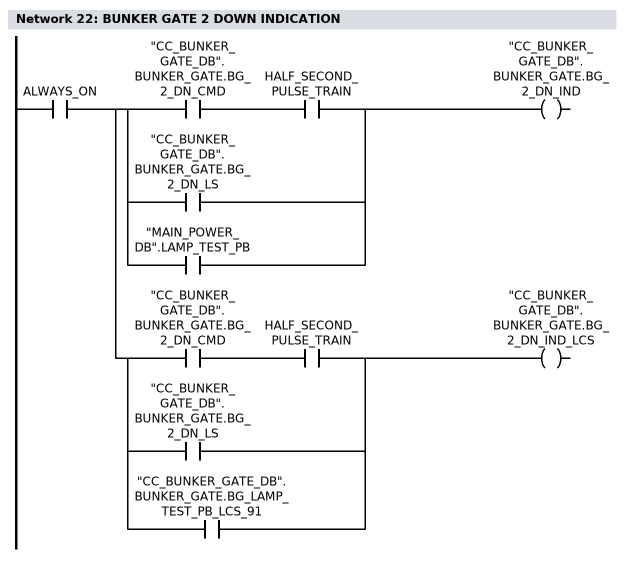
NETWORK
TITLE = BUNKER GATE 2 DOWN INDICATION
      A     "ALWAYS_ON";
      =     L 0.0;
      A     L 0.0;
      A(;
      A     "CC_BUNKER_GATE_DB".BUNKER_GATE.BG_2_DN_CMD;
      A     "HALF_SECOND_PULSE_TRAIN";
      O     "CC_BUNKER_GATE_DB".BUNKER_GATE.BG_2_DN_LS;
      O     "MAIN_POWER_DB".LAMP_TEST_PB;
      );
      =     "CC_BUNKER_GATE_DB".BUNKER_GATE.BG_2_DN_IND;
      A     L 0.0;
      A(;
      A     "CC_BUNKER_GATE_DB".BUNKER_GATE.BG_2_DN_CMD;
      A     "HALF_SECOND_PULSE_TRAIN";
      O     "CC_BUNKER_GATE_DB".BUNKER_GATE.BG_2_DN_LS;
      O     "CC_BUNKER_GATE_DB".BUNKER_GATE.BG_LAMP_TEST_PB_LCS_91;
      );
      =     "CC_BUNKER_GATE_DB".BUNKER_GATE.BG_2_DN_IND_LCS;
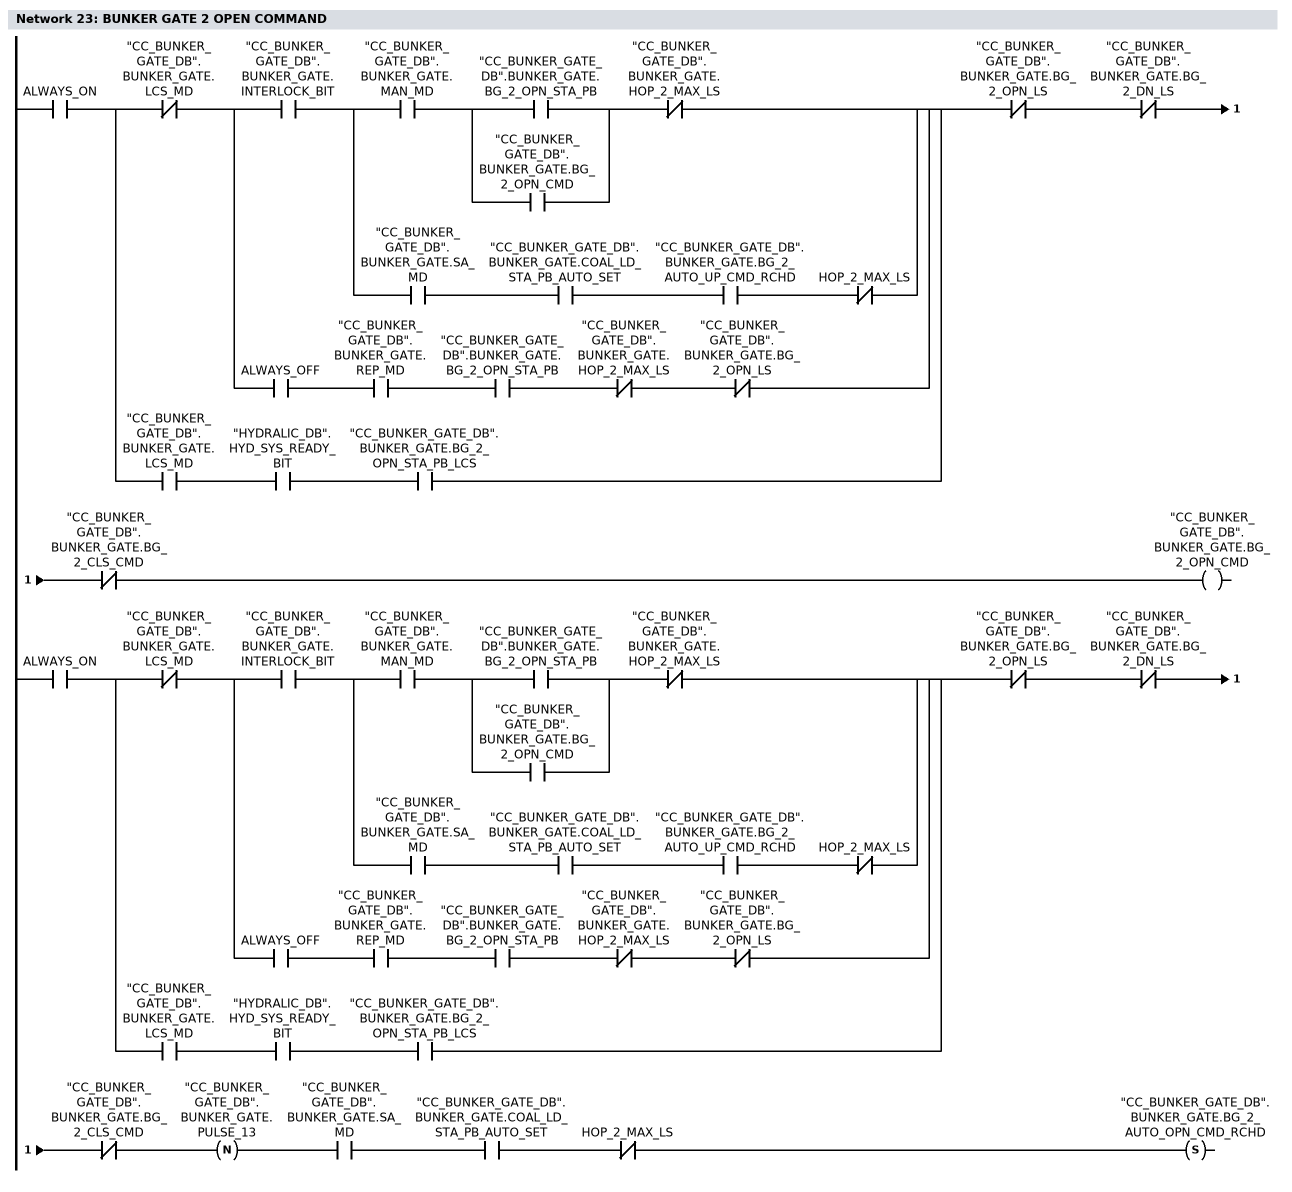
NETWORK
TITLE = BUNKER GATE 2 OPEN COMMAND
      A     "ALWAYS_ON";
      A(;
      AN    "CC_BUNKER_GATE_DB".BUNKER_GATE.LCS_MD;
      A(;
      A     "CC_BUNKER_GATE_DB".BUNKER_GATE.INTERLOCK_BIT;
      A(;
      A     "CC_BUNKER_GATE_DB".BUNKER_GATE.MAN_MD;
      A(;
      O     "CC_BUNKER_GATE_DB".BUNKER_GATE.BG_2_OPN_STA_PB;
      O     "CC_BUNKER_GATE_DB".BUNKER_GATE.BG_2_OPN_CMD;
      );
      AN    "CC_BUNKER_GATE_DB".BUNKER_GATE.HOP_2_MAX_LS;
      O;
      A     "CC_BUNKER_GATE_DB".BUNKER_GATE.SA_MD;
      A     "CC_BUNKER_GATE_DB".BUNKER_GATE.COAL_LD_STA_PB_AUTO_SET;
      A     "CC_BUNKER_GATE_DB".BUNKER_GATE.BG_2_AUTO_UP_CMD_RCHD;
      AN    "HOP_2_MAX_LS";
      );
      O;
      A     "ALWAYS_OFF";
      A     "CC_BUNKER_GATE_DB".BUNKER_GATE.REP_MD;
      A     "CC_BUNKER_GATE_DB".BUNKER_GATE.BG_2_OPN_STA_PB;
      AN    "CC_BUNKER_GATE_DB".BUNKER_GATE.HOP_2_MAX_LS;
      AN    "CC_BUNKER_GATE_DB".BUNKER_GATE.BG_2_OPN_LS;
      );
      O;
      A     "CC_BUNKER_GATE_DB".BUNKER_GATE.LCS_MD;
      A     "HYDRALIC_DB".HYD_SYS_READY_BIT;
      A     "CC_BUNKER_GATE_DB".BUNKER_GATE.BG_2_OPN_STA_PB_LCS;
      );
      AN    "CC_BUNKER_GATE_DB".BUNKER_GATE.BG_2_OPN_LS;
      AN    "CC_BUNKER_GATE_DB".BUNKER_GATE.BG_2_DN_LS;
      AN    "CC_BUNKER_GATE_DB".BUNKER_GATE.BG_2_CLS_CMD;
      =     L 0.0;
      A     L 0.0;
      BLD   102;
      =     "CC_BUNKER_GATE_DB".BUNKER_GATE.BG_2_OPN_CMD;
      A(;
      A     L 0.0;
      FN    "CC_BUNKER_GATE_DB".BUNKER_GATE.PULSE_13;
      );
      A     "CC_BUNKER_GATE_DB".BUNKER_GATE.SA_MD;
      A     "CC_BUNKER_GATE_DB".BUNKER_GATE.COAL_LD_STA_PB_AUTO_SET;
      AN    "HOP_2_MAX_LS";
      S     "CC_BUNKER_GATE_DB".BUNKER_GATE.BG_2_AUTO_OPN_CMD_RCHD;
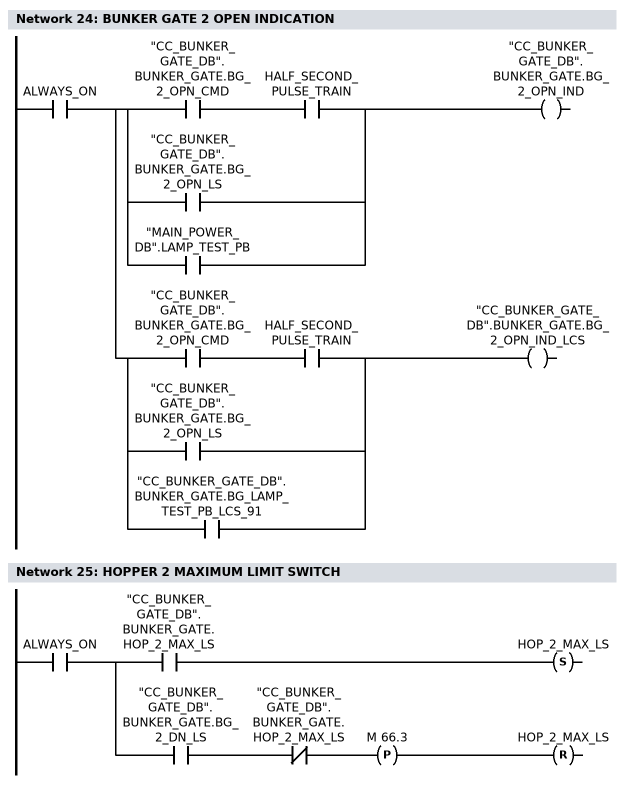
NETWORK
TITLE = BUNKER GATE 2 OPEN INDICATION
      A     "ALWAYS_ON";
      =     L 0.0;
      A     L 0.0;
      A(;
      A     "CC_BUNKER_GATE_DB".BUNKER_GATE.BG_2_OPN_CMD;
      A     "HALF_SECOND_PULSE_TRAIN";
      O     "CC_BUNKER_GATE_DB".BUNKER_GATE.BG_2_OPN_LS;
      O     "MAIN_POWER_DB".LAMP_TEST_PB;
      );
      =     "CC_BUNKER_GATE_DB".BUNKER_GATE.BG_2_OPN_IND;
      A     L 0.0;
      A(;
      A     "CC_BUNKER_GATE_DB".BUNKER_GATE.BG_2_OPN_CMD;
      A     "HALF_SECOND_PULSE_TRAIN";
      O     "CC_BUNKER_GATE_DB".BUNKER_GATE.BG_2_OPN_LS;
      O     "CC_BUNKER_GATE_DB".BUNKER_GATE.BG_LAMP_TEST_PB_LCS_91;
      );
      =     "CC_BUNKER_GATE_DB".BUNKER_GATE.BG_2_OPN_IND_LCS;
NETWORK
TITLE = HOPPER 2 MAXIMUM LIMIT SWITCH
      A     "ALWAYS_ON";
      =     L 0.0;
      A     L 0.0;
      A     "CC_BUNKER_GATE_DB".BUNKER_GATE.HOP_2_MAX_LS;
      S     "HOP_2_MAX_LS";
      A     L 0.0;
      A     "CC_BUNKER_GATE_DB".BUNKER_GATE.BG_2_DN_LS;
      AN    "CC_BUNKER_GATE_DB".BUNKER_GATE.HOP_2_MAX_LS;
      FP    M 66.3;
      R     "HOP_2_MAX_LS";
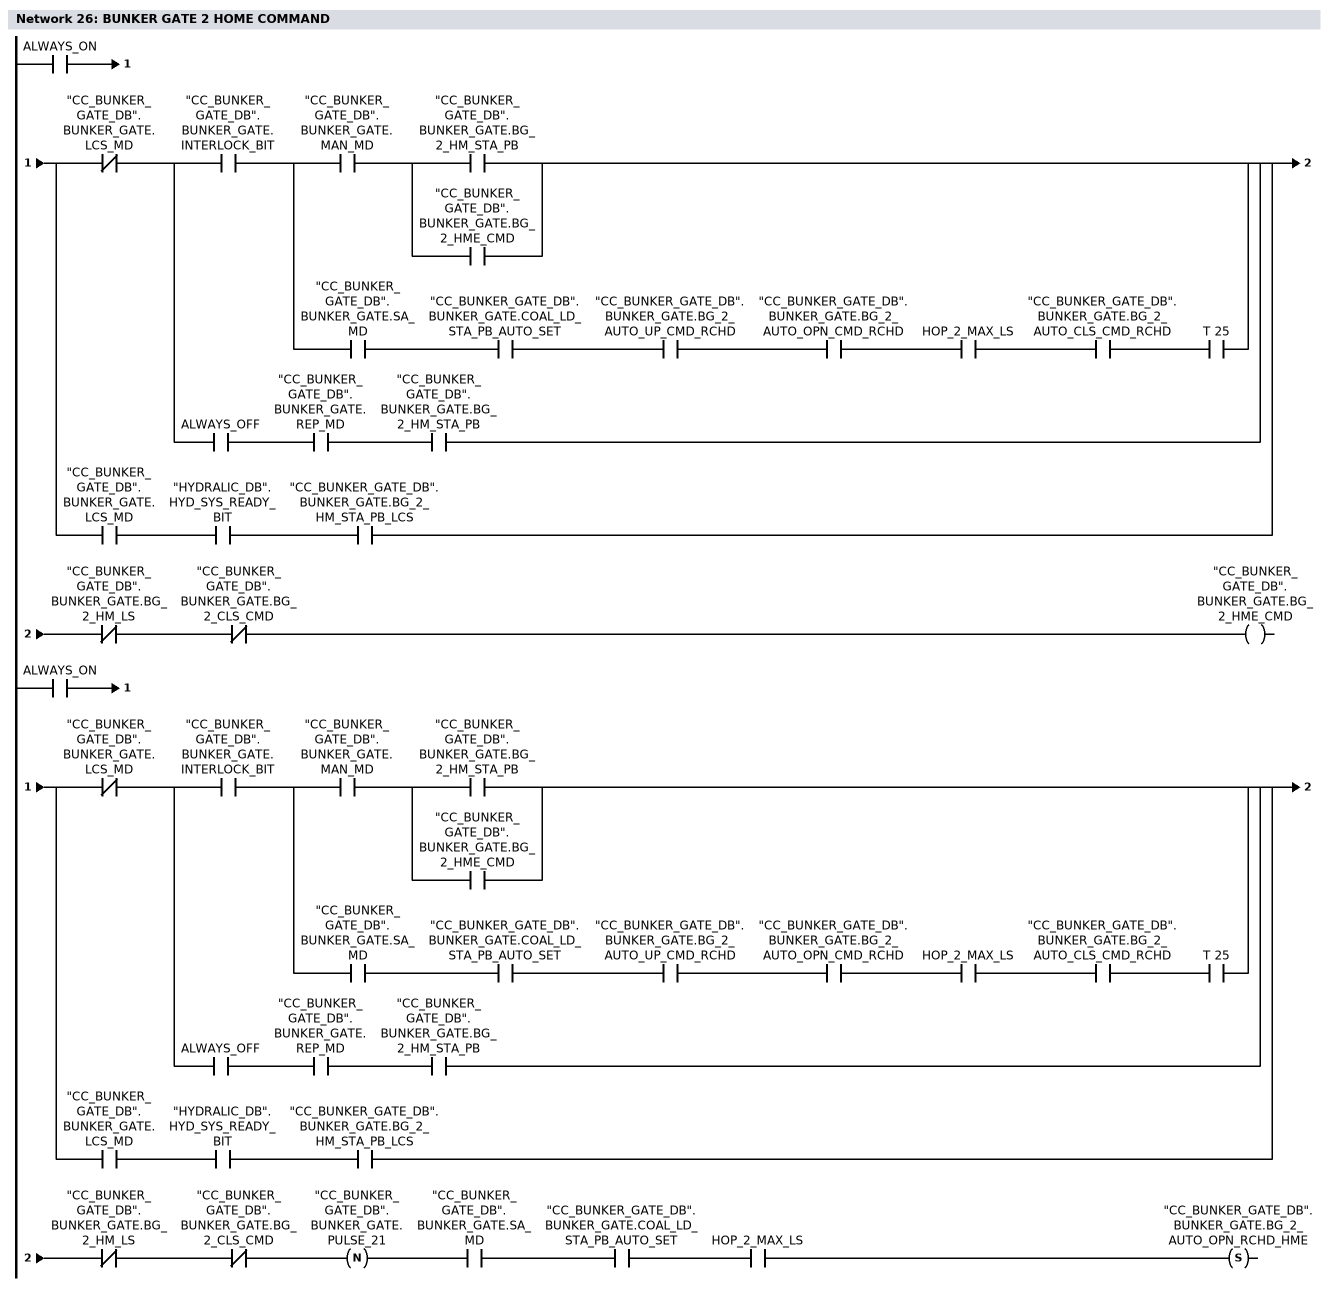
NETWORK
TITLE = BUNKER GATE 2 HOME COMMAND
      A     "ALWAYS_ON";
      A(;
      AN    "CC_BUNKER_GATE_DB".BUNKER_GATE.LCS_MD;
      A(;
      A     "CC_BUNKER_GATE_DB".BUNKER_GATE.INTERLOCK_BIT;
      A(;
      A     "CC_BUNKER_GATE_DB".BUNKER_GATE.MAN_MD;
      A(;
      O     "CC_BUNKER_GATE_DB".BUNKER_GATE.BG_2_HM_STA_PB;
      O     "CC_BUNKER_GATE_DB".BUNKER_GATE.BG_2_HME_CMD;
      );
      O;
      A     "CC_BUNKER_GATE_DB".BUNKER_GATE.SA_MD;
      A     "CC_BUNKER_GATE_DB".BUNKER_GATE.COAL_LD_STA_PB_AUTO_SET;
      A     "CC_BUNKER_GATE_DB".BUNKER_GATE.BG_2_AUTO_UP_CMD_RCHD;
      A     "CC_BUNKER_GATE_DB".BUNKER_GATE.BG_2_AUTO_OPN_CMD_RCHD;
      A     "HOP_2_MAX_LS";
      A     "CC_BUNKER_GATE_DB".BUNKER_GATE.BG_2_AUTO_CLS_CMD_RCHD;
      A     T 25;
      );
      O;
      A     "ALWAYS_OFF";
      A     "CC_BUNKER_GATE_DB".BUNKER_GATE.REP_MD;
      A     "CC_BUNKER_GATE_DB".BUNKER_GATE.BG_2_HM_STA_PB;
      );
      O;
      A     "CC_BUNKER_GATE_DB".BUNKER_GATE.LCS_MD;
      A     "HYDRALIC_DB".HYD_SYS_READY_BIT;
      A     "CC_BUNKER_GATE_DB".BUNKER_GATE.BG_2_HM_STA_PB_LCS;
      );
      AN    "CC_BUNKER_GATE_DB".BUNKER_GATE.BG_2_HM_LS;
      AN    "CC_BUNKER_GATE_DB".BUNKER_GATE.BG_2_CLS_CMD;
      =     L 0.0;
      A     L 0.0;
      BLD   102;
      =     "CC_BUNKER_GATE_DB".BUNKER_GATE.BG_2_HME_CMD;
      A(;
      A     L 0.0;
      FN    "CC_BUNKER_GATE_DB".BUNKER_GATE.PULSE_21;
      );
      A     "CC_BUNKER_GATE_DB".BUNKER_GATE.SA_MD;
      A     "CC_BUNKER_GATE_DB".BUNKER_GATE.COAL_LD_STA_PB_AUTO_SET;
      A     "HOP_2_MAX_LS";
      S     "CC_BUNKER_GATE_DB".BUNKER_GATE.BG_2_AUTO_OPN_RCHD_HME;
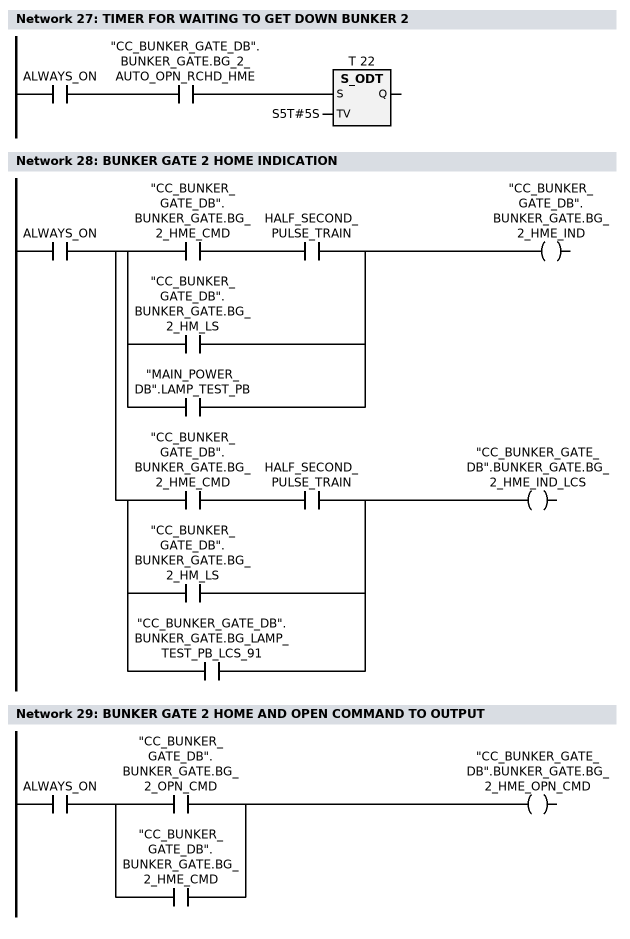
NETWORK
TITLE = TIMER FOR WAITING TO GET DOWN BUNKER 2
      A     "ALWAYS_ON";
      A     "CC_BUNKER_GATE_DB".BUNKER_GATE.BG_2_AUTO_OPN_RCHD_HME;
      L     S5T#5S;
      SD    T 22;
      NOP   0;
      NOP   0;
      NOP   0;
      NOP   0;
NETWORK
TITLE = BUNKER GATE 2 HOME INDICATION
      A     "ALWAYS_ON";
      =     L 0.0;
      A     L 0.0;
      A(;
      A     "CC_BUNKER_GATE_DB".BUNKER_GATE.BG_2_HME_CMD;
      A     "HALF_SECOND_PULSE_TRAIN";
      O     "CC_BUNKER_GATE_DB".BUNKER_GATE.BG_2_HM_LS;
      O     "MAIN_POWER_DB".LAMP_TEST_PB;
      );
      =     "CC_BUNKER_GATE_DB".BUNKER_GATE.BG_2_HME_IND;
      A     L 0.0;
      A(;
      A     "CC_BUNKER_GATE_DB".BUNKER_GATE.BG_2_HME_CMD;
      A     "HALF_SECOND_PULSE_TRAIN";
      O     "CC_BUNKER_GATE_DB".BUNKER_GATE.BG_2_HM_LS;
      O     "CC_BUNKER_GATE_DB".BUNKER_GATE.BG_LAMP_TEST_PB_LCS_91;
      );
      =     "CC_BUNKER_GATE_DB".BUNKER_GATE.BG_2_HME_IND_LCS;
NETWORK
TITLE = BUNKER GATE 2 HOME AND OPEN COMMAND TO OUTPUT
      A     "ALWAYS_ON";
      A(;
      O     "CC_BUNKER_GATE_DB".BUNKER_GATE.BG_2_OPN_CMD;
      O     "CC_BUNKER_GATE_DB".BUNKER_GATE.BG_2_HME_CMD;
      );
      =     "CC_BUNKER_GATE_DB".BUNKER_GATE.BG_2_HME_OPN_CMD;
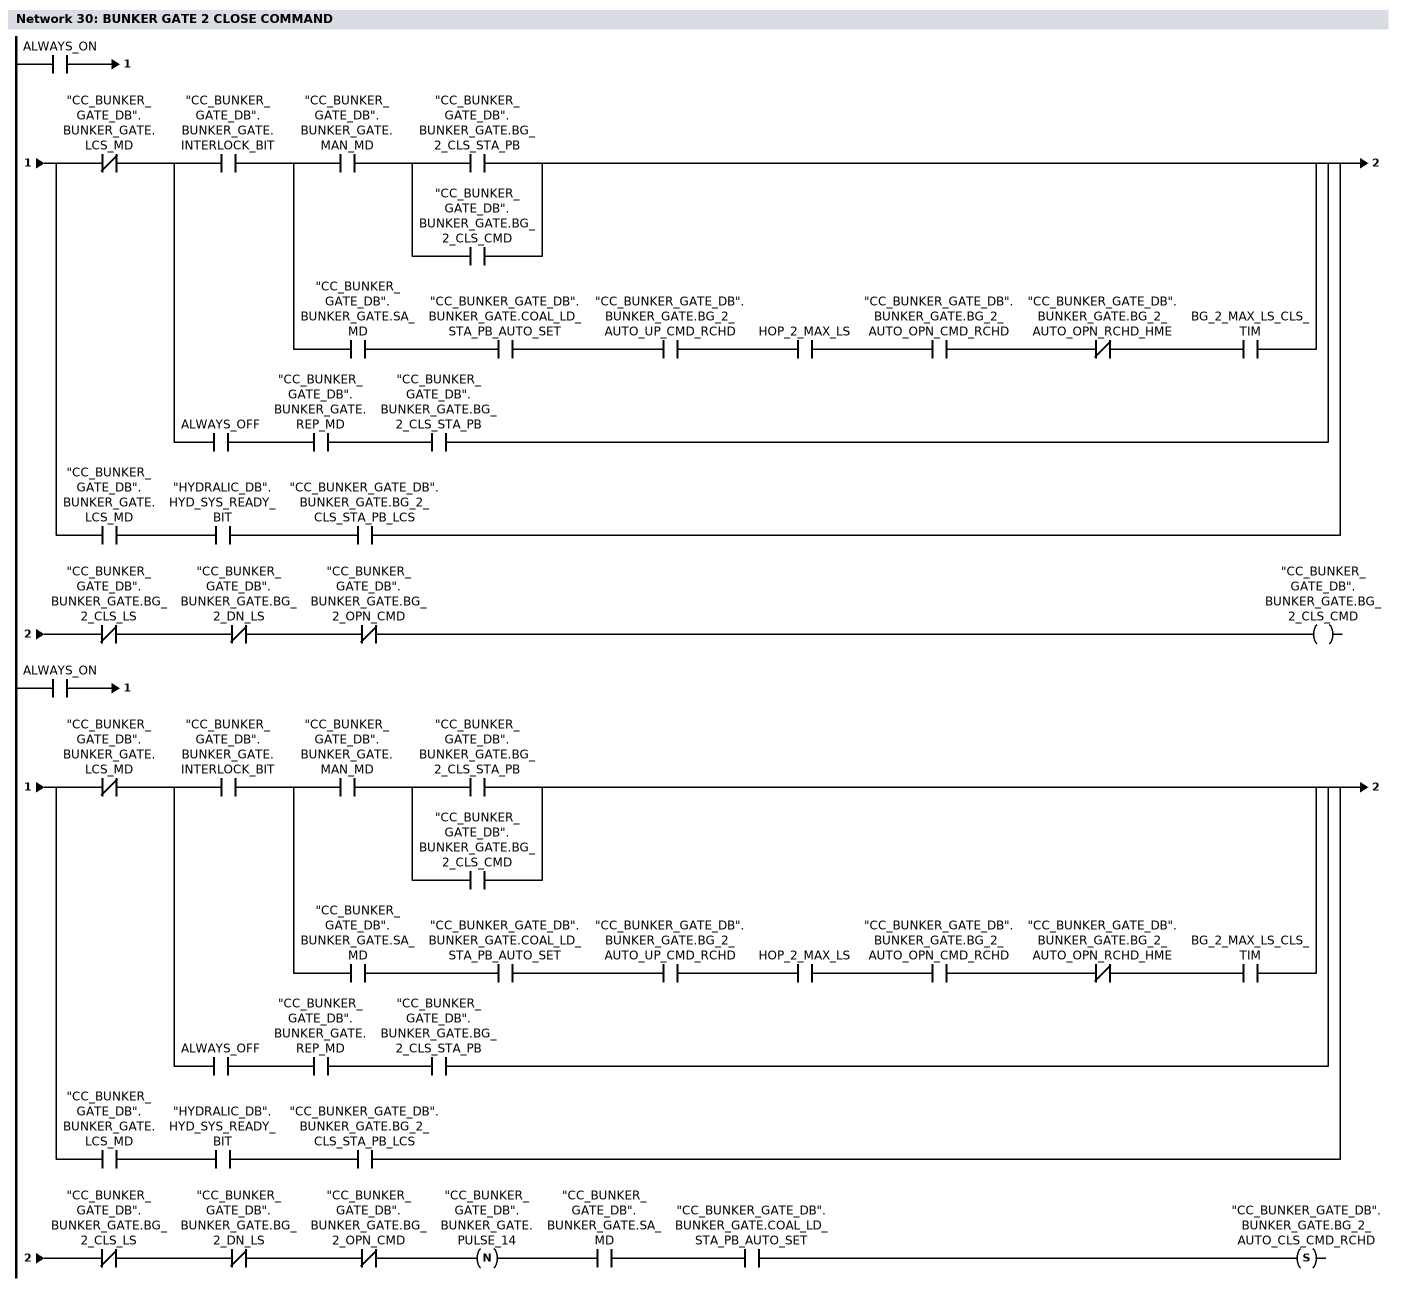
NETWORK
TITLE = BUNKER GATE 2 CLOSE COMMAND
      A     "ALWAYS_ON";
      A(;
      AN    "CC_BUNKER_GATE_DB".BUNKER_GATE.LCS_MD;
      A(;
      A     "CC_BUNKER_GATE_DB".BUNKER_GATE.INTERLOCK_BIT;
      A(;
      A     "CC_BUNKER_GATE_DB".BUNKER_GATE.MAN_MD;
      A(;
      O     "CC_BUNKER_GATE_DB".BUNKER_GATE.BG_2_CLS_STA_PB;
      O     "CC_BUNKER_GATE_DB".BUNKER_GATE.BG_2_CLS_CMD;
      );
      O;
      A     "CC_BUNKER_GATE_DB".BUNKER_GATE.SA_MD;
      A     "CC_BUNKER_GATE_DB".BUNKER_GATE.COAL_LD_STA_PB_AUTO_SET;
      A     "CC_BUNKER_GATE_DB".BUNKER_GATE.BG_2_AUTO_UP_CMD_RCHD;
      A     "HOP_2_MAX_LS";
      A     "CC_BUNKER_GATE_DB".BUNKER_GATE.BG_2_AUTO_OPN_CMD_RCHD;
      AN    "CC_BUNKER_GATE_DB".BUNKER_GATE.BG_2_AUTO_OPN_RCHD_HME;
      A     "BG_2_MAX_LS_CLS_TIM";
      );
      O;
      A     "ALWAYS_OFF";
      A     "CC_BUNKER_GATE_DB".BUNKER_GATE.REP_MD;
      A     "CC_BUNKER_GATE_DB".BUNKER_GATE.BG_2_CLS_STA_PB;
      );
      O;
      A     "CC_BUNKER_GATE_DB".BUNKER_GATE.LCS_MD;
      A     "HYDRALIC_DB".HYD_SYS_READY_BIT;
      A     "CC_BUNKER_GATE_DB".BUNKER_GATE.BG_2_CLS_STA_PB_LCS;
      );
      AN    "CC_BUNKER_GATE_DB".BUNKER_GATE.BG_2_CLS_LS;
      AN    "CC_BUNKER_GATE_DB".BUNKER_GATE.BG_2_DN_LS;
      AN    "CC_BUNKER_GATE_DB".BUNKER_GATE.BG_2_OPN_CMD;
      =     L 0.0;
      A     L 0.0;
      BLD   102;
      =     "CC_BUNKER_GATE_DB".BUNKER_GATE.BG_2_CLS_CMD;
      A(;
      A     L 0.0;
      FN    "CC_BUNKER_GATE_DB".BUNKER_GATE.PULSE_14;
      );
      A     "CC_BUNKER_GATE_DB".BUNKER_GATE.SA_MD;
      A     "CC_BUNKER_GATE_DB".BUNKER_GATE.COAL_LD_STA_PB_AUTO_SET;
      S     "CC_BUNKER_GATE_DB".BUNKER_GATE.BG_2_AUTO_CLS_CMD_RCHD;
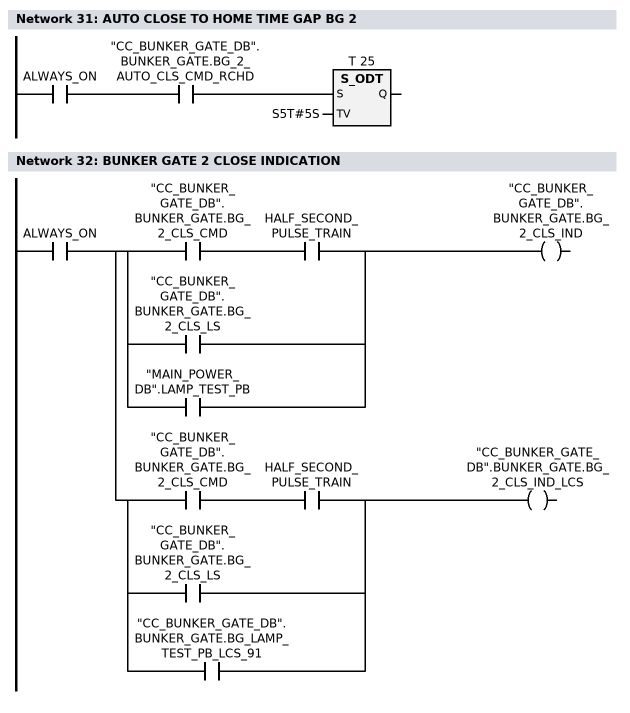
NETWORK
TITLE = AUTO CLOSE TO HOME TIME GAP BG 2
      A     "ALWAYS_ON";
      A     "CC_BUNKER_GATE_DB".BUNKER_GATE.BG_2_AUTO_CLS_CMD_RCHD;
      L     S5T#5S;
      SD    T 25;
      NOP   0;
      NOP   0;
      NOP   0;
      NOP   0;
NETWORK
TITLE = BUNKER GATE 2 CLOSE INDICATION
      A     "ALWAYS_ON";
      =     L 0.0;
      A     L 0.0;
      A(;
      A     "CC_BUNKER_GATE_DB".BUNKER_GATE.BG_2_CLS_CMD;
      A     "HALF_SECOND_PULSE_TRAIN";
      O     "CC_BUNKER_GATE_DB".BUNKER_GATE.BG_2_CLS_LS;
      O     "MAIN_POWER_DB".LAMP_TEST_PB;
      );
      =     "CC_BUNKER_GATE_DB".BUNKER_GATE.BG_2_CLS_IND;
      A     L 0.0;
      A(;
      A     "CC_BUNKER_GATE_DB".BUNKER_GATE.BG_2_CLS_CMD;
      A     "HALF_SECOND_PULSE_TRAIN";
      O     "CC_BUNKER_GATE_DB".BUNKER_GATE.BG_2_CLS_LS;
      O     "CC_BUNKER_GATE_DB".BUNKER_GATE.BG_LAMP_TEST_PB_LCS_91;
      );
      =     "CC_BUNKER_GATE_DB".BUNKER_GATE.BG_2_CLS_IND_LCS;
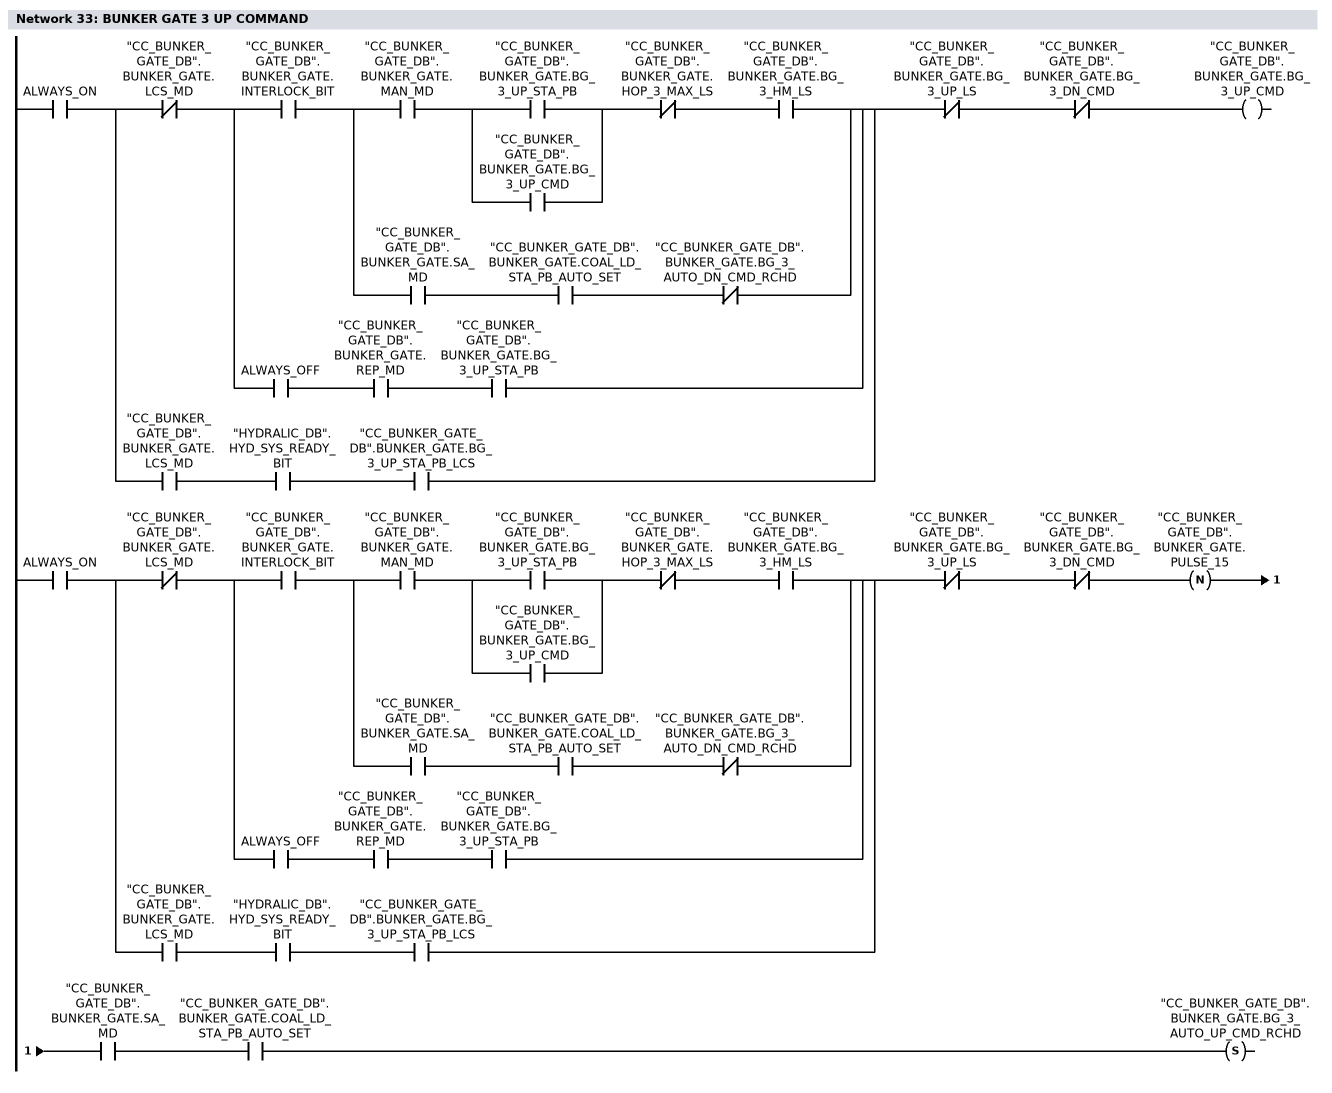
NETWORK
TITLE = BUNKER GATE 3 UP COMMAND
      A     "ALWAYS_ON";
      A(;
      AN    "CC_BUNKER_GATE_DB".BUNKER_GATE.LCS_MD;
      A(;
      A     "CC_BUNKER_GATE_DB".BUNKER_GATE.INTERLOCK_BIT;
      A(;
      A     "CC_BUNKER_GATE_DB".BUNKER_GATE.MAN_MD;
      A(;
      O     "CC_BUNKER_GATE_DB".BUNKER_GATE.BG_3_UP_STA_PB;
      O     "CC_BUNKER_GATE_DB".BUNKER_GATE.BG_3_UP_CMD;
      );
      AN    "CC_BUNKER_GATE_DB".BUNKER_GATE.HOP_3_MAX_LS;
      A     "CC_BUNKER_GATE_DB".BUNKER_GATE.BG_3_HM_LS;
      O;
      A     "CC_BUNKER_GATE_DB".BUNKER_GATE.SA_MD;
      A     "CC_BUNKER_GATE_DB".BUNKER_GATE.COAL_LD_STA_PB_AUTO_SET;
      AN    "CC_BUNKER_GATE_DB".BUNKER_GATE.BG_3_AUTO_DN_CMD_RCHD;
      );
      O;
      A     "ALWAYS_OFF";
      A     "CC_BUNKER_GATE_DB".BUNKER_GATE.REP_MD;
      A     "CC_BUNKER_GATE_DB".BUNKER_GATE.BG_3_UP_STA_PB;
      );
      O;
      A     "CC_BUNKER_GATE_DB".BUNKER_GATE.LCS_MD;
      A     "HYDRALIC_DB".HYD_SYS_READY_BIT;
      A     "CC_BUNKER_GATE_DB".BUNKER_GATE.BG_3_UP_STA_PB_LCS;
      );
      AN    "CC_BUNKER_GATE_DB".BUNKER_GATE.BG_3_UP_LS;
      AN    "CC_BUNKER_GATE_DB".BUNKER_GATE.BG_3_DN_CMD;
      =     L 0.0;
      A     L 0.0;
      BLD   102;
      =     "CC_BUNKER_GATE_DB".BUNKER_GATE.BG_3_UP_CMD;
      A(;
      A     L 0.0;
      FN    "CC_BUNKER_GATE_DB".BUNKER_GATE.PULSE_15;
      );
      A     "CC_BUNKER_GATE_DB".BUNKER_GATE.SA_MD;
      A     "CC_BUNKER_GATE_DB".BUNKER_GATE.COAL_LD_STA_PB_AUTO_SET;
      S     "CC_BUNKER_GATE_DB".BUNKER_GATE.BG_3_AUTO_UP_CMD_RCHD;
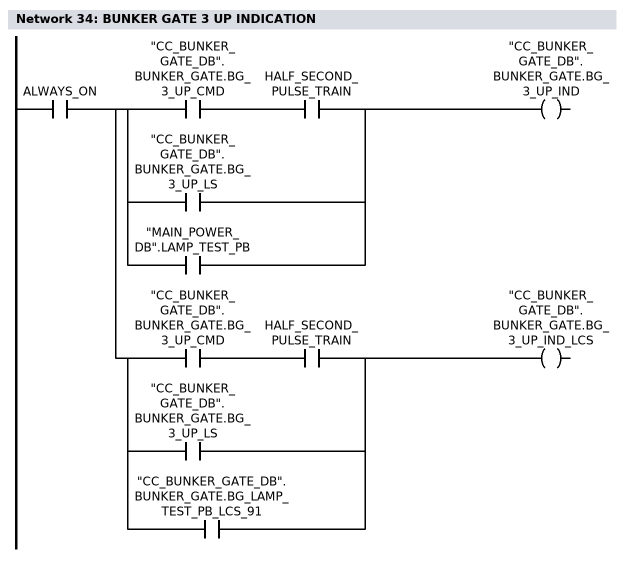
NETWORK
TITLE = BUNKER GATE 3 UP INDICATION
      A     "ALWAYS_ON";
      =     L 0.0;
      A     L 0.0;
      A(;
      A     "CC_BUNKER_GATE_DB".BUNKER_GATE.BG_3_UP_CMD;
      A     "HALF_SECOND_PULSE_TRAIN";
      O     "CC_BUNKER_GATE_DB".BUNKER_GATE.BG_3_UP_LS;
      O     "MAIN_POWER_DB".LAMP_TEST_PB;
      );
      =     "CC_BUNKER_GATE_DB".BUNKER_GATE.BG_3_UP_IND;
      A     L 0.0;
      A(;
      A     "CC_BUNKER_GATE_DB".BUNKER_GATE.BG_3_UP_CMD;
      A     "HALF_SECOND_PULSE_TRAIN";
      O     "CC_BUNKER_GATE_DB".BUNKER_GATE.BG_3_UP_LS;
      O     "CC_BUNKER_GATE_DB".BUNKER_GATE.BG_LAMP_TEST_PB_LCS_91;
      );
      =     "CC_BUNKER_GATE_DB".BUNKER_GATE.BG_3_UP_IND_LCS;
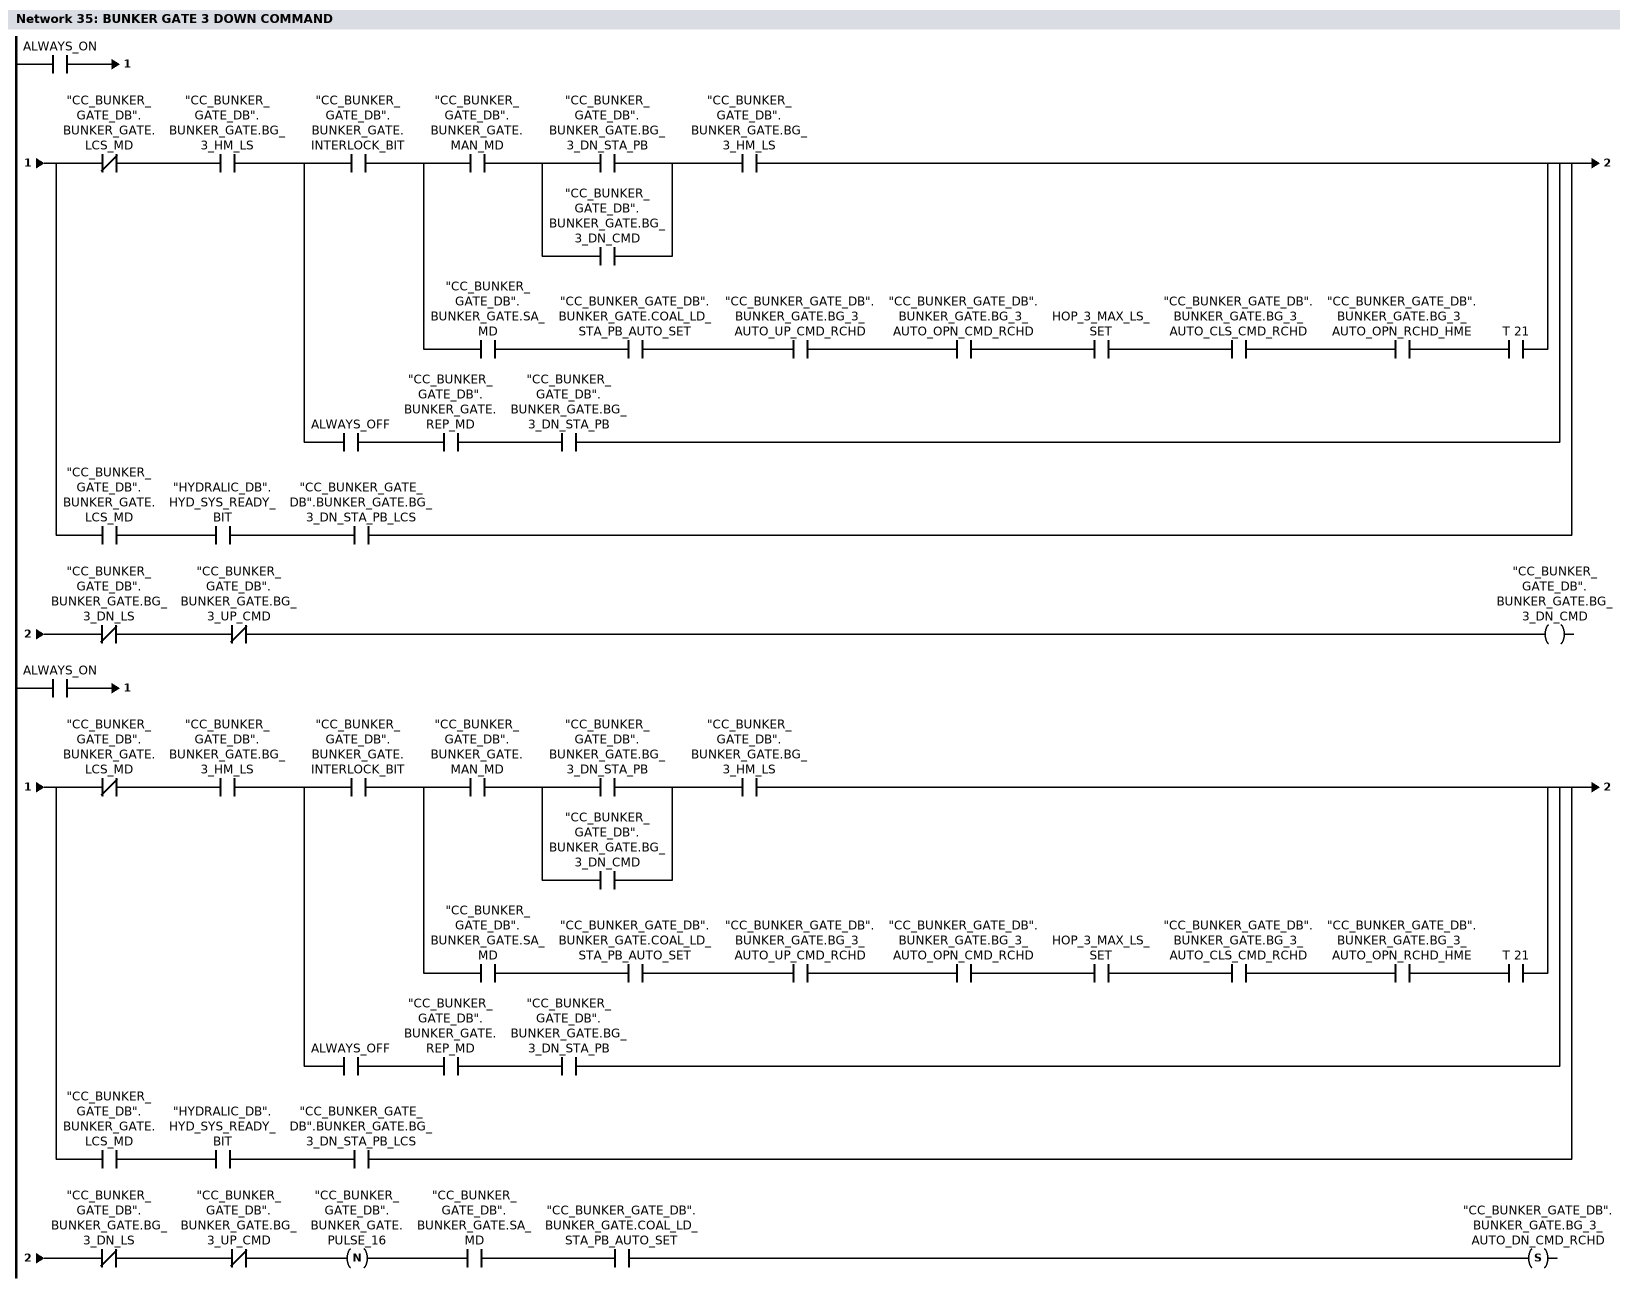
NETWORK
TITLE = BUNKER GATE 3 DOWN COMMAND
      A     "ALWAYS_ON";
      A(;
      AN    "CC_BUNKER_GATE_DB".BUNKER_GATE.LCS_MD;
      A     "CC_BUNKER_GATE_DB".BUNKER_GATE.BG_3_HM_LS;
      A(;
      A     "CC_BUNKER_GATE_DB".BUNKER_GATE.INTERLOCK_BIT;
      A(;
      A     "CC_BUNKER_GATE_DB".BUNKER_GATE.MAN_MD;
      A(;
      O     "CC_BUNKER_GATE_DB".BUNKER_GATE.BG_3_DN_STA_PB;
      O     "CC_BUNKER_GATE_DB".BUNKER_GATE.BG_3_DN_CMD;
      );
      A     "CC_BUNKER_GATE_DB".BUNKER_GATE.BG_3_HM_LS;
      O;
      A     "CC_BUNKER_GATE_DB".BUNKER_GATE.SA_MD;
      A     "CC_BUNKER_GATE_DB".BUNKER_GATE.COAL_LD_STA_PB_AUTO_SET;
      A     "CC_BUNKER_GATE_DB".BUNKER_GATE.BG_3_AUTO_UP_CMD_RCHD;
      A     "CC_BUNKER_GATE_DB".BUNKER_GATE.BG_3_AUTO_OPN_CMD_RCHD;
      A     "HOP_3_MAX_LS_SET";
      A     "CC_BUNKER_GATE_DB".BUNKER_GATE.BG_3_AUTO_CLS_CMD_RCHD;
      A     "CC_BUNKER_GATE_DB".BUNKER_GATE.BG_3_AUTO_OPN_RCHD_HME;
      A     T 21;
      );
      O;
      A     "ALWAYS_OFF";
      A     "CC_BUNKER_GATE_DB".BUNKER_GATE.REP_MD;
      A     "CC_BUNKER_GATE_DB".BUNKER_GATE.BG_3_DN_STA_PB;
      );
      O;
      A     "CC_BUNKER_GATE_DB".BUNKER_GATE.LCS_MD;
      A     "HYDRALIC_DB".HYD_SYS_READY_BIT;
      A     "CC_BUNKER_GATE_DB".BUNKER_GATE.BG_3_DN_STA_PB_LCS;
      );
      AN    "CC_BUNKER_GATE_DB".BUNKER_GATE.BG_3_DN_LS;
      AN    "CC_BUNKER_GATE_DB".BUNKER_GATE.BG_3_UP_CMD;
      =     L 0.0;
      A     L 0.0;
      BLD   102;
      =     "CC_BUNKER_GATE_DB".BUNKER_GATE.BG_3_DN_CMD;
      A(;
      A     L 0.0;
      FN    "CC_BUNKER_GATE_DB".BUNKER_GATE.PULSE_16;
      );
      A     "CC_BUNKER_GATE_DB".BUNKER_GATE.SA_MD;
      A     "CC_BUNKER_GATE_DB".BUNKER_GATE.COAL_LD_STA_PB_AUTO_SET;
      S     "CC_BUNKER_GATE_DB".BUNKER_GATE.BG_3_AUTO_DN_CMD_RCHD;
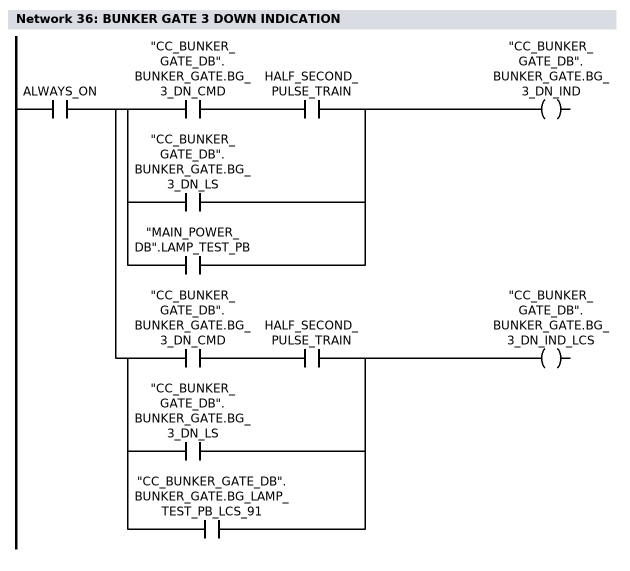
NETWORK
TITLE = BUNKER GATE 3 DOWN INDICATION
      A     "ALWAYS_ON";
      =     L 0.0;
      A     L 0.0;
      A(;
      A     "CC_BUNKER_GATE_DB".BUNKER_GATE.BG_3_DN_CMD;
      A     "HALF_SECOND_PULSE_TRAIN";
      O     "CC_BUNKER_GATE_DB".BUNKER_GATE.BG_3_DN_LS;
      O     "MAIN_POWER_DB".LAMP_TEST_PB;
      );
      =     "CC_BUNKER_GATE_DB".BUNKER_GATE.BG_3_DN_IND;
      A     L 0.0;
      A(;
      A     "CC_BUNKER_GATE_DB".BUNKER_GATE.BG_3_DN_CMD;
      A     "HALF_SECOND_PULSE_TRAIN";
      O     "CC_BUNKER_GATE_DB".BUNKER_GATE.BG_3_DN_LS;
      O     "CC_BUNKER_GATE_DB".BUNKER_GATE.BG_LAMP_TEST_PB_LCS_91;
      );
      =     "CC_BUNKER_GATE_DB".BUNKER_GATE.BG_3_DN_IND_LCS;
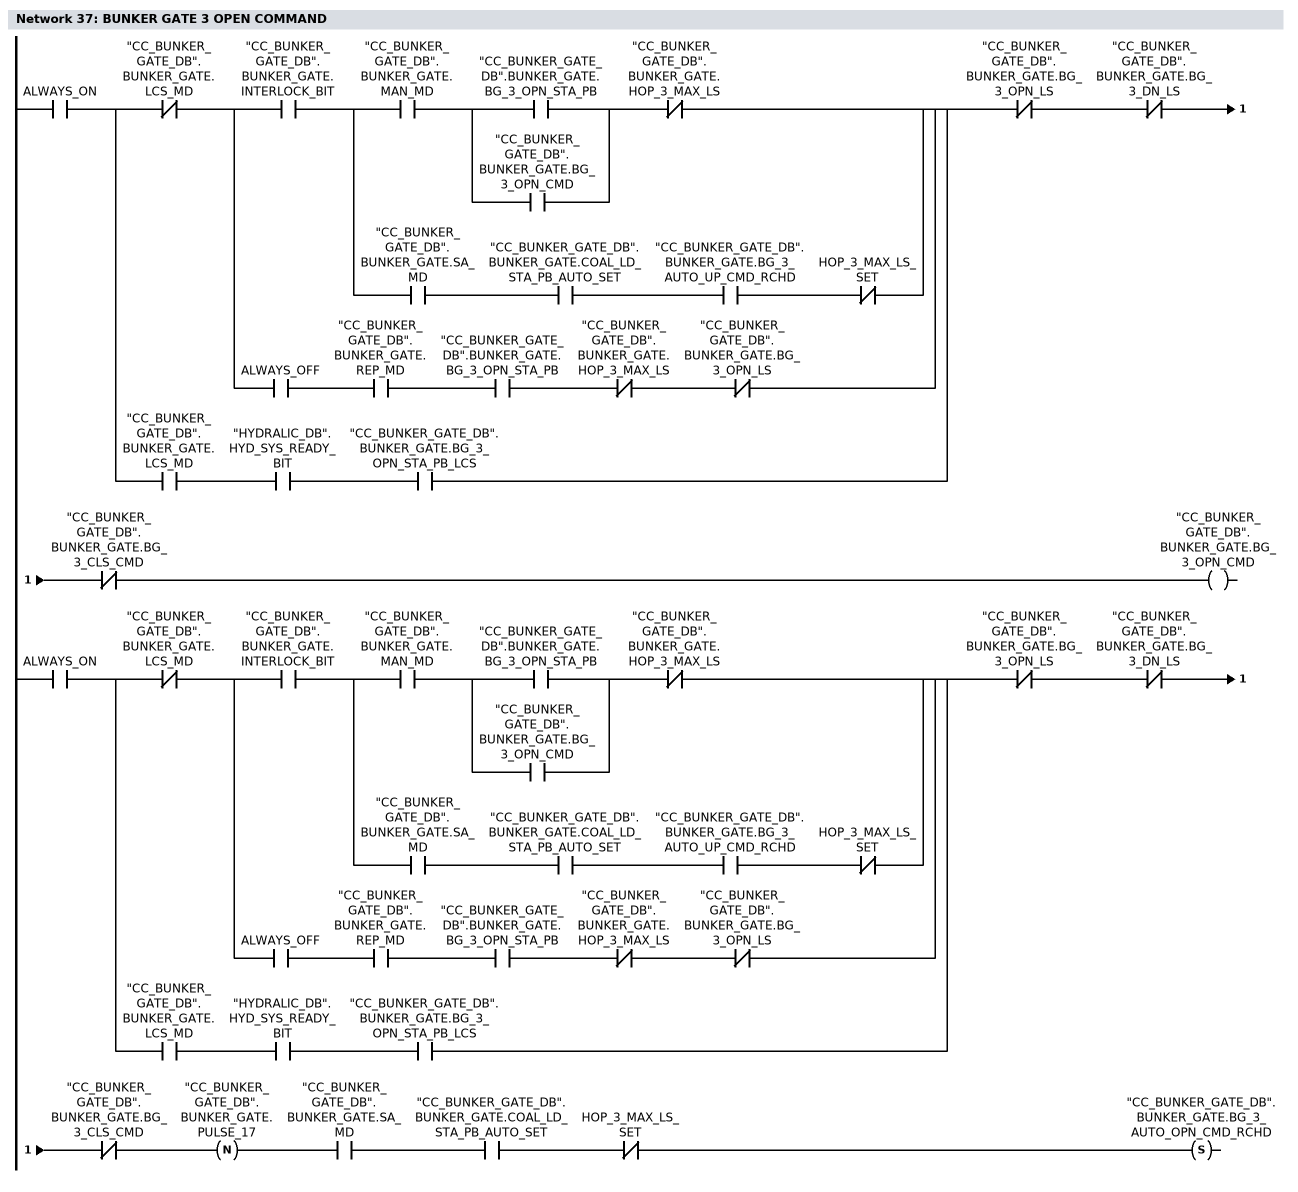
NETWORK
TITLE = BUNKER GATE 3 OPEN COMMAND
      A     "ALWAYS_ON";
      A(;
      AN    "CC_BUNKER_GATE_DB".BUNKER_GATE.LCS_MD;
      A(;
      A     "CC_BUNKER_GATE_DB".BUNKER_GATE.INTERLOCK_BIT;
      A(;
      A     "CC_BUNKER_GATE_DB".BUNKER_GATE.MAN_MD;
      A(;
      O     "CC_BUNKER_GATE_DB".BUNKER_GATE.BG_3_OPN_STA_PB;
      O     "CC_BUNKER_GATE_DB".BUNKER_GATE.BG_3_OPN_CMD;
      );
      AN    "CC_BUNKER_GATE_DB".BUNKER_GATE.HOP_3_MAX_LS;
      O;
      A     "CC_BUNKER_GATE_DB".BUNKER_GATE.SA_MD;
      A     "CC_BUNKER_GATE_DB".BUNKER_GATE.COAL_LD_STA_PB_AUTO_SET;
      A     "CC_BUNKER_GATE_DB".BUNKER_GATE.BG_3_AUTO_UP_CMD_RCHD;
      AN    "HOP_3_MAX_LS_SET";
      );
      O;
      A     "ALWAYS_OFF";
      A     "CC_BUNKER_GATE_DB".BUNKER_GATE.REP_MD;
      A     "CC_BUNKER_GATE_DB".BUNKER_GATE.BG_3_OPN_STA_PB;
      AN    "CC_BUNKER_GATE_DB".BUNKER_GATE.HOP_3_MAX_LS;
      AN    "CC_BUNKER_GATE_DB".BUNKER_GATE.BG_3_OPN_LS;
      );
      O;
      A     "CC_BUNKER_GATE_DB".BUNKER_GATE.LCS_MD;
      A     "HYDRALIC_DB".HYD_SYS_READY_BIT;
      A     "CC_BUNKER_GATE_DB".BUNKER_GATE.BG_3_OPN_STA_PB_LCS;
      );
      AN    "CC_BUNKER_GATE_DB".BUNKER_GATE.BG_3_OPN_LS;
      AN    "CC_BUNKER_GATE_DB".BUNKER_GATE.BG_3_DN_LS;
      AN    "CC_BUNKER_GATE_DB".BUNKER_GATE.BG_3_CLS_CMD;
      =     L 0.0;
      A     L 0.0;
      BLD   102;
      =     "CC_BUNKER_GATE_DB".BUNKER_GATE.BG_3_OPN_CMD;
      A(;
      A     L 0.0;
      FN    "CC_BUNKER_GATE_DB".BUNKER_GATE.PULSE_17;
      );
      A     "CC_BUNKER_GATE_DB".BUNKER_GATE.SA_MD;
      A     "CC_BUNKER_GATE_DB".BUNKER_GATE.COAL_LD_STA_PB_AUTO_SET;
      AN    "HOP_3_MAX_LS_SET";
      S     "CC_BUNKER_GATE_DB".BUNKER_GATE.BG_3_AUTO_OPN_CMD_RCHD;
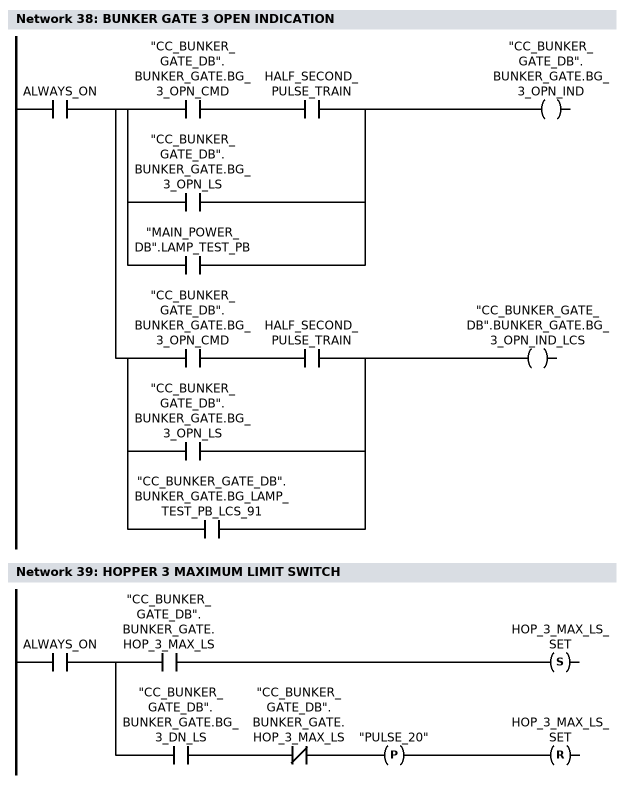
NETWORK
TITLE = BUNKER GATE 3 OPEN INDICATION
      A     "ALWAYS_ON";
      =     L 0.0;
      A     L 0.0;
      A(;
      A     "CC_BUNKER_GATE_DB".BUNKER_GATE.BG_3_OPN_CMD;
      A     "HALF_SECOND_PULSE_TRAIN";
      O     "CC_BUNKER_GATE_DB".BUNKER_GATE.BG_3_OPN_LS;
      O     "MAIN_POWER_DB".LAMP_TEST_PB;
      );
      =     "CC_BUNKER_GATE_DB".BUNKER_GATE.BG_3_OPN_IND;
      A     L 0.0;
      A(;
      A     "CC_BUNKER_GATE_DB".BUNKER_GATE.BG_3_OPN_CMD;
      A     "HALF_SECOND_PULSE_TRAIN";
      O     "CC_BUNKER_GATE_DB".BUNKER_GATE.BG_3_OPN_LS;
      O     "CC_BUNKER_GATE_DB".BUNKER_GATE.BG_LAMP_TEST_PB_LCS_91;
      );
      =     "CC_BUNKER_GATE_DB".BUNKER_GATE.BG_3_OPN_IND_LCS;
NETWORK
TITLE = HOPPER 3 MAXIMUM LIMIT SWITCH
      A     "ALWAYS_ON";
      =     L 0.0;
      A     L 0.0;
      A     "CC_BUNKER_GATE_DB".BUNKER_GATE.HOP_3_MAX_LS;
      S     "HOP_3_MAX_LS_SET";
      A     L 0.0;
      A     "CC_BUNKER_GATE_DB".BUNKER_GATE.BG_3_DN_LS;
      AN    "CC_BUNKER_GATE_DB".BUNKER_GATE.HOP_3_MAX_LS;
      FP    "PULSE_20";
      R     "HOP_3_MAX_LS_SET";
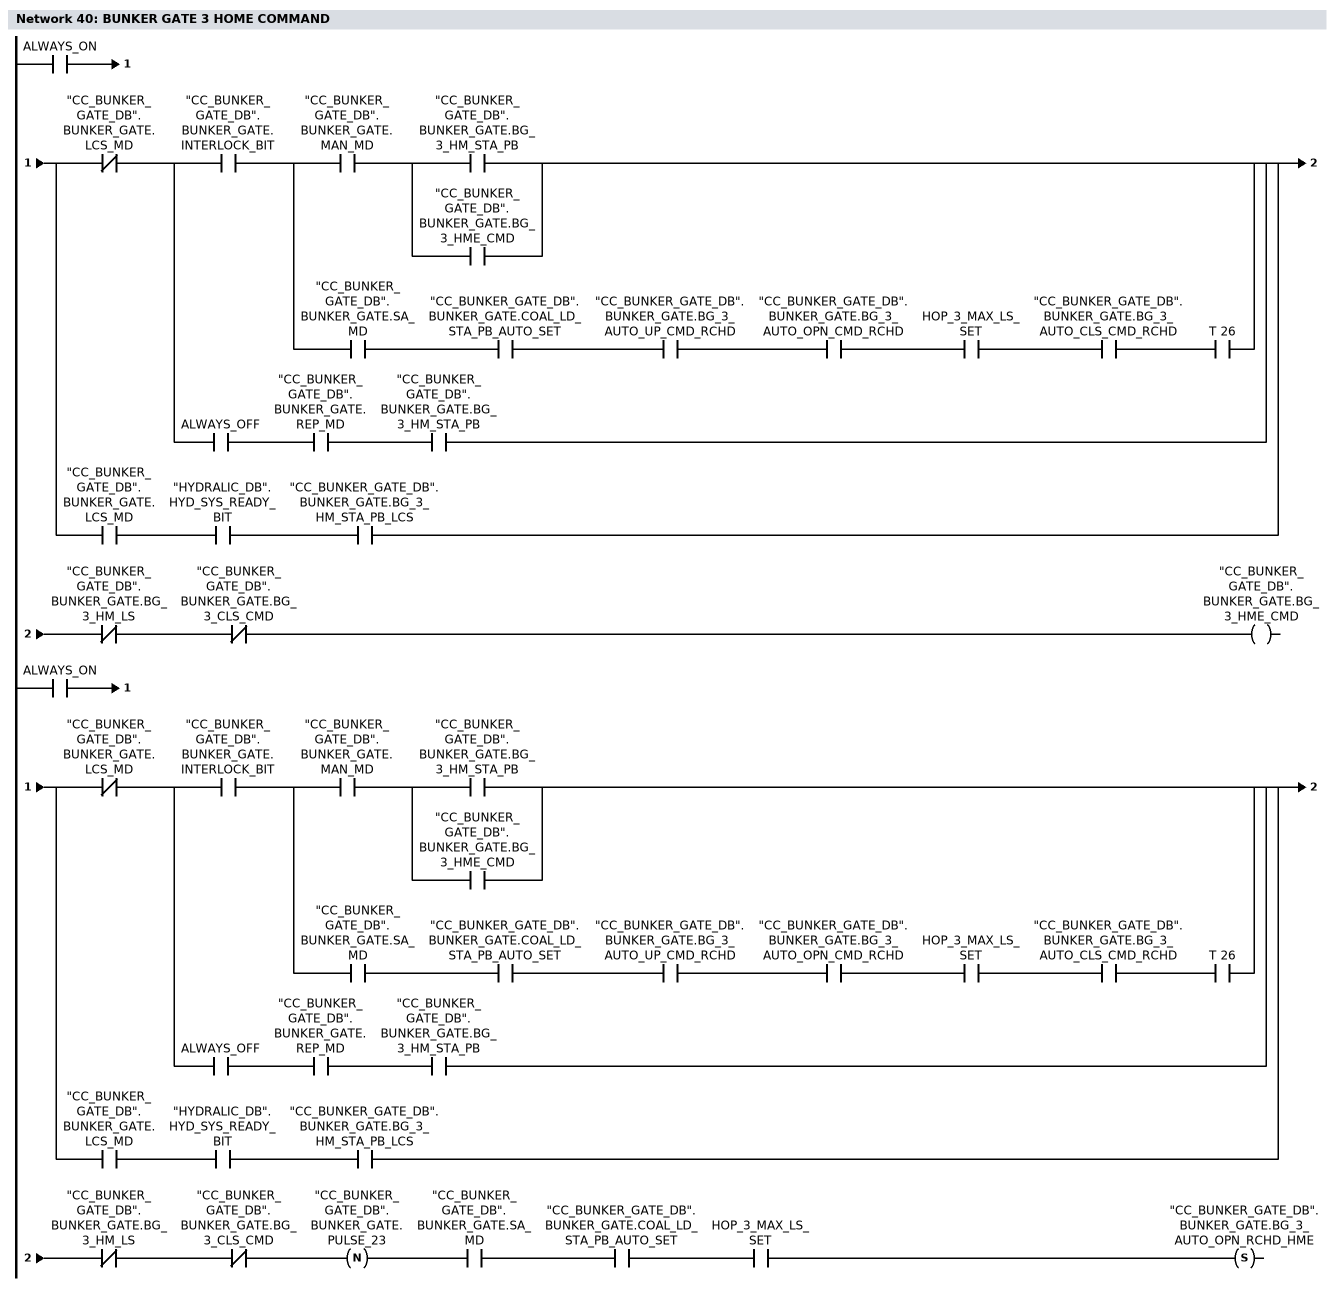
NETWORK
TITLE = BUNKER GATE 3 HOME COMMAND
      A     "ALWAYS_ON";
      A(;
      AN    "CC_BUNKER_GATE_DB".BUNKER_GATE.LCS_MD;
      A(;
      A     "CC_BUNKER_GATE_DB".BUNKER_GATE.INTERLOCK_BIT;
      A(;
      A     "CC_BUNKER_GATE_DB".BUNKER_GATE.MAN_MD;
      A(;
      O     "CC_BUNKER_GATE_DB".BUNKER_GATE.BG_3_HM_STA_PB;
      O     "CC_BUNKER_GATE_DB".BUNKER_GATE.BG_3_HME_CMD;
      );
      O;
      A     "CC_BUNKER_GATE_DB".BUNKER_GATE.SA_MD;
      A     "CC_BUNKER_GATE_DB".BUNKER_GATE.COAL_LD_STA_PB_AUTO_SET;
      A     "CC_BUNKER_GATE_DB".BUNKER_GATE.BG_3_AUTO_UP_CMD_RCHD;
      A     "CC_BUNKER_GATE_DB".BUNKER_GATE.BG_3_AUTO_OPN_CMD_RCHD;
      A     "HOP_3_MAX_LS_SET";
      A     "CC_BUNKER_GATE_DB".BUNKER_GATE.BG_3_AUTO_CLS_CMD_RCHD;
      A     T 26;
      );
      O;
      A     "ALWAYS_OFF";
      A     "CC_BUNKER_GATE_DB".BUNKER_GATE.REP_MD;
      A     "CC_BUNKER_GATE_DB".BUNKER_GATE.BG_3_HM_STA_PB;
      );
      O;
      A     "CC_BUNKER_GATE_DB".BUNKER_GATE.LCS_MD;
      A     "HYDRALIC_DB".HYD_SYS_READY_BIT;
      A     "CC_BUNKER_GATE_DB".BUNKER_GATE.BG_3_HM_STA_PB_LCS;
      );
      AN    "CC_BUNKER_GATE_DB".BUNKER_GATE.BG_3_HM_LS;
      AN    "CC_BUNKER_GATE_DB".BUNKER_GATE.BG_3_CLS_CMD;
      =     L 0.0;
      A     L 0.0;
      BLD   102;
      =     "CC_BUNKER_GATE_DB".BUNKER_GATE.BG_3_HME_CMD;
      A(;
      A     L 0.0;
      FN    "CC_BUNKER_GATE_DB".BUNKER_GATE.PULSE_23;
      );
      A     "CC_BUNKER_GATE_DB".BUNKER_GATE.SA_MD;
      A     "CC_BUNKER_GATE_DB".BUNKER_GATE.COAL_LD_STA_PB_AUTO_SET;
      A     "HOP_3_MAX_LS_SET";
      S     "CC_BUNKER_GATE_DB".BUNKER_GATE.BG_3_AUTO_OPN_RCHD_HME;
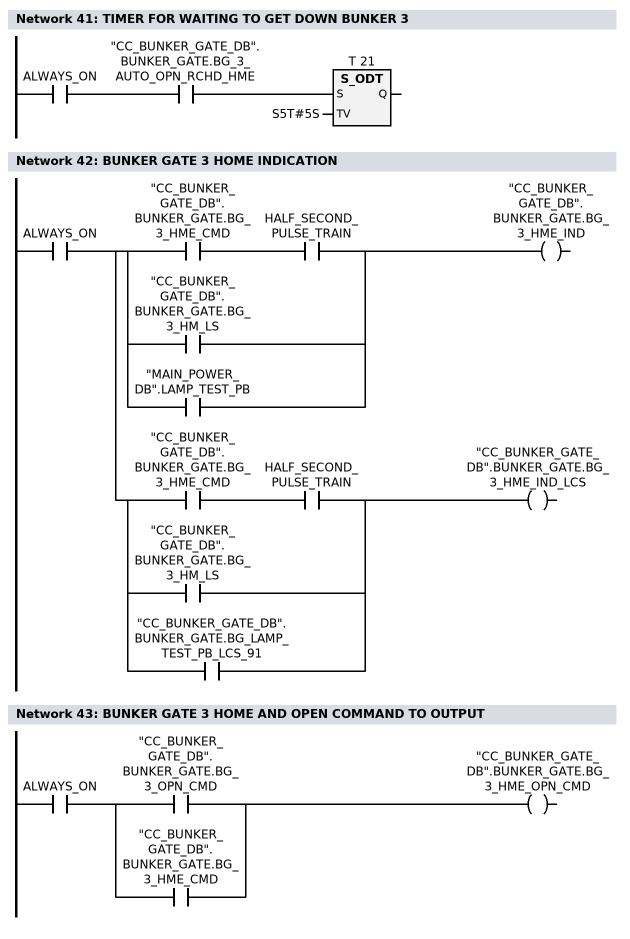
NETWORK
TITLE = TIMER FOR WAITING TO GET DOWN BUNKER 3
      A     "ALWAYS_ON";
      A     "CC_BUNKER_GATE_DB".BUNKER_GATE.BG_3_AUTO_OPN_RCHD_HME;
      L     S5T#5S;
      SD    T 21;
      NOP   0;
      NOP   0;
      NOP   0;
      NOP   0;
NETWORK
TITLE = BUNKER GATE 3 HOME INDICATION
      A     "ALWAYS_ON";
      =     L 0.0;
      A     L 0.0;
      A(;
      A     "CC_BUNKER_GATE_DB".BUNKER_GATE.BG_3_HME_CMD;
      A     "HALF_SECOND_PULSE_TRAIN";
      O     "CC_BUNKER_GATE_DB".BUNKER_GATE.BG_3_HM_LS;
      O     "MAIN_POWER_DB".LAMP_TEST_PB;
      );
      =     "CC_BUNKER_GATE_DB".BUNKER_GATE.BG_3_HME_IND;
      A     L 0.0;
      A(;
      A     "CC_BUNKER_GATE_DB".BUNKER_GATE.BG_3_HME_CMD;
      A     "HALF_SECOND_PULSE_TRAIN";
      O     "CC_BUNKER_GATE_DB".BUNKER_GATE.BG_3_HM_LS;
      O     "CC_BUNKER_GATE_DB".BUNKER_GATE.BG_LAMP_TEST_PB_LCS_91;
      );
      =     "CC_BUNKER_GATE_DB".BUNKER_GATE.BG_3_HME_IND_LCS;
NETWORK
TITLE = BUNKER GATE 3 HOME AND OPEN COMMAND TO OUTPUT
      A     "ALWAYS_ON";
      A(;
      O     "CC_BUNKER_GATE_DB".BUNKER_GATE.BG_3_OPN_CMD;
      O     "CC_BUNKER_GATE_DB".BUNKER_GATE.BG_3_HME_CMD;
      );
      =     "CC_BUNKER_GATE_DB".BUNKER_GATE.BG_3_HME_OPN_CMD;
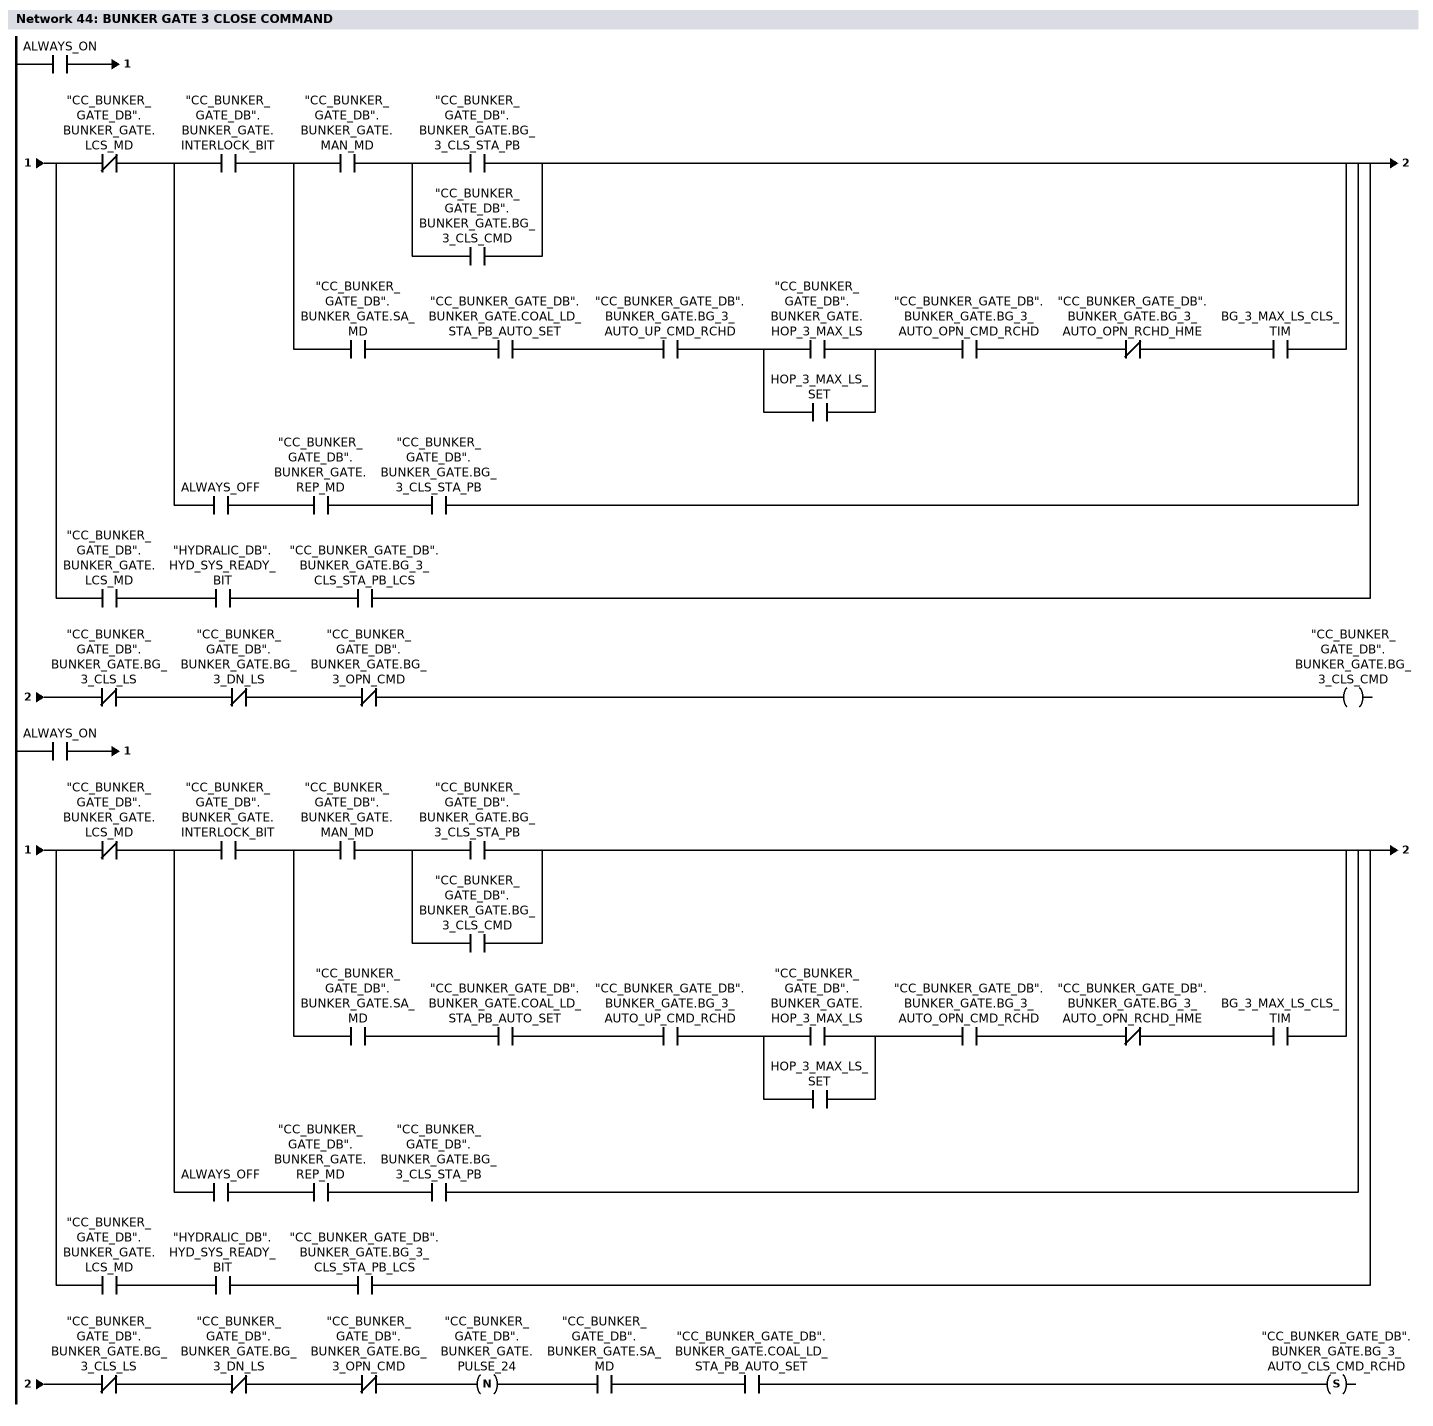
NETWORK
TITLE = BUNKER GATE 3 CLOSE COMMAND
      A     "ALWAYS_ON";
      A(;
      AN    "CC_BUNKER_GATE_DB".BUNKER_GATE.LCS_MD;
      A(;
      A     "CC_BUNKER_GATE_DB".BUNKER_GATE.INTERLOCK_BIT;
      A(;
      A     "CC_BUNKER_GATE_DB".BUNKER_GATE.MAN_MD;
      A(;
      O     "CC_BUNKER_GATE_DB".BUNKER_GATE.BG_3_CLS_STA_PB;
      O     "CC_BUNKER_GATE_DB".BUNKER_GATE.BG_3_CLS_CMD;
      );
      O;
      A     "CC_BUNKER_GATE_DB".BUNKER_GATE.SA_MD;
      A     "CC_BUNKER_GATE_DB".BUNKER_GATE.COAL_LD_STA_PB_AUTO_SET;
      A     "CC_BUNKER_GATE_DB".BUNKER_GATE.BG_3_AUTO_UP_CMD_RCHD;
      A(;
      O     "CC_BUNKER_GATE_DB".BUNKER_GATE.HOP_3_MAX_LS;
      O     "HOP_3_MAX_LS_SET";
      );
      A     "CC_BUNKER_GATE_DB".BUNKER_GATE.BG_3_AUTO_OPN_CMD_RCHD;
      AN    "CC_BUNKER_GATE_DB".BUNKER_GATE.BG_3_AUTO_OPN_RCHD_HME;
      A     "BG_3_MAX_LS_CLS_TIM";
      );
      O;
      A     "ALWAYS_OFF";
      A     "CC_BUNKER_GATE_DB".BUNKER_GATE.REP_MD;
      A     "CC_BUNKER_GATE_DB".BUNKER_GATE.BG_3_CLS_STA_PB;
      );
      O;
      A     "CC_BUNKER_GATE_DB".BUNKER_GATE.LCS_MD;
      A     "HYDRALIC_DB".HYD_SYS_READY_BIT;
      A     "CC_BUNKER_GATE_DB".BUNKER_GATE.BG_3_CLS_STA_PB_LCS;
      );
      AN    "CC_BUNKER_GATE_DB".BUNKER_GATE.BG_3_CLS_LS;
      AN    "CC_BUNKER_GATE_DB".BUNKER_GATE.BG_3_DN_LS;
      AN    "CC_BUNKER_GATE_DB".BUNKER_GATE.BG_3_OPN_CMD;
      =     L 0.0;
      A     L 0.0;
      BLD   102;
      =     "CC_BUNKER_GATE_DB".BUNKER_GATE.BG_3_CLS_CMD;
      A(;
      A     L 0.0;
      FN    "CC_BUNKER_GATE_DB".BUNKER_GATE.PULSE_24;
      );
      A     "CC_BUNKER_GATE_DB".BUNKER_GATE.SA_MD;
      A     "CC_BUNKER_GATE_DB".BUNKER_GATE.COAL_LD_STA_PB_AUTO_SET;
      S     "CC_BUNKER_GATE_DB".BUNKER_GATE.BG_3_AUTO_CLS_CMD_RCHD;
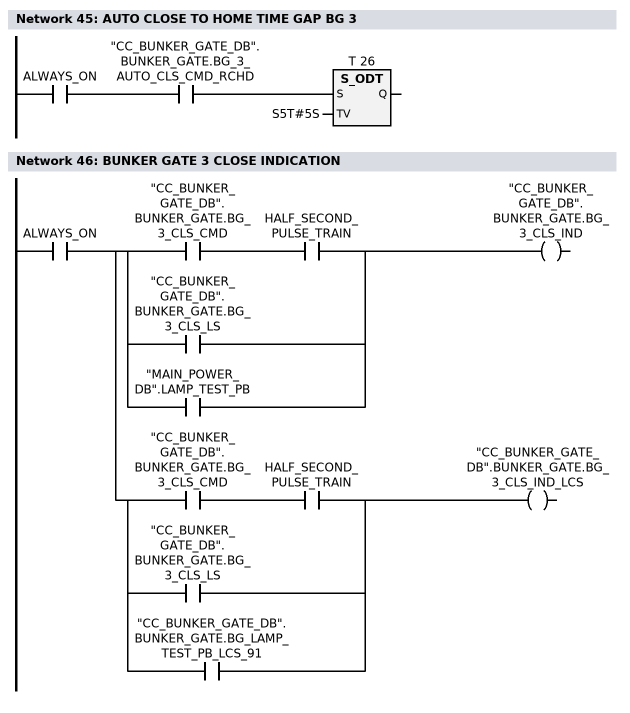
NETWORK
TITLE = AUTO CLOSE TO HOME TIME GAP BG 3
      A     "ALWAYS_ON";
      A     "CC_BUNKER_GATE_DB".BUNKER_GATE.BG_3_AUTO_CLS_CMD_RCHD;
      L     S5T#5S;
      SD    T 26;
      NOP   0;
      NOP   0;
      NOP   0;
      NOP   0;
NETWORK
TITLE = BUNKER GATE 3 CLOSE INDICATION
      A     "ALWAYS_ON";
      =     L 0.0;
      A     L 0.0;
      A(;
      A     "CC_BUNKER_GATE_DB".BUNKER_GATE.BG_3_CLS_CMD;
      A     "HALF_SECOND_PULSE_TRAIN";
      O     "CC_BUNKER_GATE_DB".BUNKER_GATE.BG_3_CLS_LS;
      O     "MAIN_POWER_DB".LAMP_TEST_PB;
      );
      =     "CC_BUNKER_GATE_DB".BUNKER_GATE.BG_3_CLS_IND;
      A     L 0.0;
      A(;
      A     "CC_BUNKER_GATE_DB".BUNKER_GATE.BG_3_CLS_CMD;
      A     "HALF_SECOND_PULSE_TRAIN";
      O     "CC_BUNKER_GATE_DB".BUNKER_GATE.BG_3_CLS_LS;
      O     "CC_BUNKER_GATE_DB".BUNKER_GATE.BG_LAMP_TEST_PB_LCS_91;
      );
      =     "CC_BUNKER_GATE_DB".BUNKER_GATE.BG_3_CLS_IND_LCS;
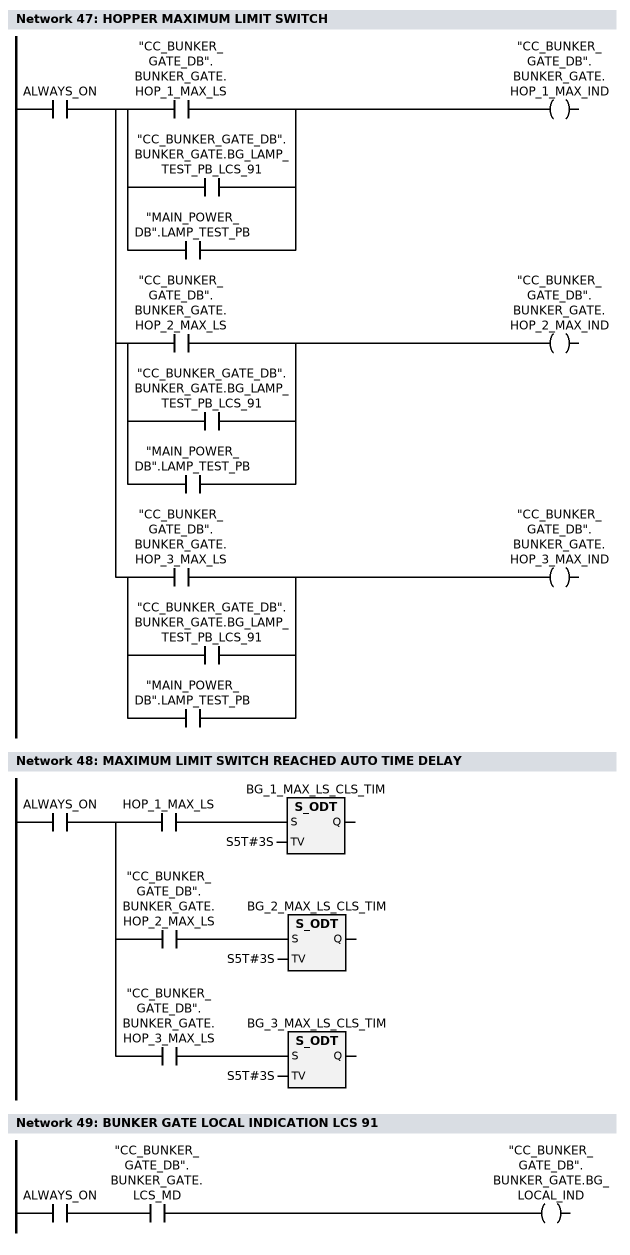
NETWORK
TITLE = HOPPER MAXIMUM LIMIT SWITCH
      A     "ALWAYS_ON";
      =     L 0.0;
      A     L 0.0;
      A(;
      O     "CC_BUNKER_GATE_DB".BUNKER_GATE.HOP_1_MAX_LS;
      O     "CC_BUNKER_GATE_DB".BUNKER_GATE.BG_LAMP_TEST_PB_LCS_91;
      O     "MAIN_POWER_DB".LAMP_TEST_PB;
      );
      =     "CC_BUNKER_GATE_DB".BUNKER_GATE.HOP_1_MAX_IND;
      A     L 0.0;
      A(;
      O     "CC_BUNKER_GATE_DB".BUNKER_GATE.HOP_2_MAX_LS;
      O     "CC_BUNKER_GATE_DB".BUNKER_GATE.BG_LAMP_TEST_PB_LCS_91;
      O     "MAIN_POWER_DB".LAMP_TEST_PB;
      );
      =     "CC_BUNKER_GATE_DB".BUNKER_GATE.HOP_2_MAX_IND;
      A     L 0.0;
      A(;
      O     "CC_BUNKER_GATE_DB".BUNKER_GATE.HOP_3_MAX_LS;
      O     "CC_BUNKER_GATE_DB".BUNKER_GATE.BG_LAMP_TEST_PB_LCS_91;
      O     "MAIN_POWER_DB".LAMP_TEST_PB;
      );
      =     "CC_BUNKER_GATE_DB".BUNKER_GATE.HOP_3_MAX_IND;
NETWORK
TITLE = MAXIMUM LIMIT SWITCH REACHED AUTO TIME DELAY
      A     "ALWAYS_ON";
      =     L 0.0;
      A     L 0.0;
      A     "HOP_1_MAX_LS";
      L     S5T#3S;
      SD    "BG_1_MAX_LS_CLS_TIM";
      NOP   0;
      NOP   0;
      NOP   0;
      NOP   0;
      A     L 0.0;
      A     "CC_BUNKER_GATE_DB".BUNKER_GATE.HOP_2_MAX_LS;
      L     S5T#3S;
      SD    "BG_2_MAX_LS_CLS_TIM";
      NOP   0;
      NOP   0;
      NOP   0;
      NOP   0;
      A     L 0.0;
      A     "CC_BUNKER_GATE_DB".BUNKER_GATE.HOP_3_MAX_LS;
      L     S5T#3S;
      SD    "BG_3_MAX_LS_CLS_TIM";
      NOP   0;
      NOP   0;
      NOP   0;
      NOP   0;
NETWORK
TITLE = BUNKER GATE LOCAL INDICATION LCS 91
      A     "ALWAYS_ON";
      A     "CC_BUNKER_GATE_DB".BUNKER_GATE.LCS_MD;
      =     "CC_BUNKER_GATE_DB".BUNKER_GATE.BG_LOCAL_IND;
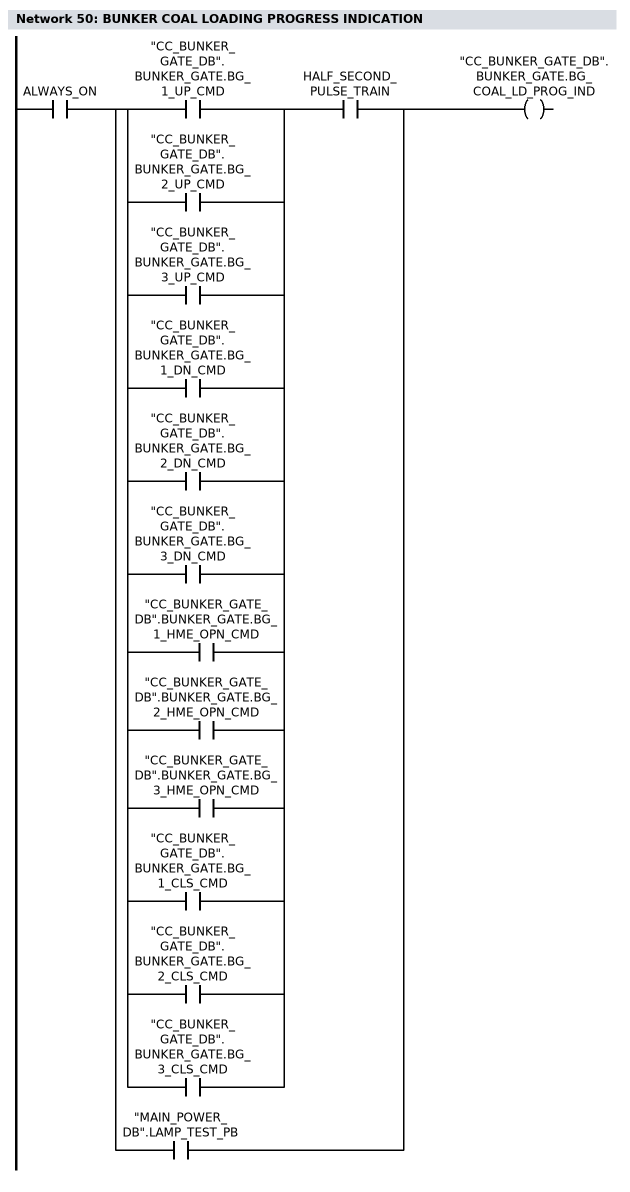
NETWORK
TITLE = BUNKER COAL LOADING PROGRESS INDICATION
      A     "ALWAYS_ON";
      A(;
      A(;
      O     "CC_BUNKER_GATE_DB".BUNKER_GATE.BG_1_UP_CMD;
      O     "CC_BUNKER_GATE_DB".BUNKER_GATE.BG_2_UP_CMD;
      O     "CC_BUNKER_GATE_DB".BUNKER_GATE.BG_3_UP_CMD;
      O     "CC_BUNKER_GATE_DB".BUNKER_GATE.BG_1_DN_CMD;
      O     "CC_BUNKER_GATE_DB".BUNKER_GATE.BG_2_DN_CMD;
      O     "CC_BUNKER_GATE_DB".BUNKER_GATE.BG_3_DN_CMD;
      O     "CC_BUNKER_GATE_DB".BUNKER_GATE.BG_1_HME_OPN_CMD;
      O     "CC_BUNKER_GATE_DB".BUNKER_GATE.BG_2_HME_OPN_CMD;
      O     "CC_BUNKER_GATE_DB".BUNKER_GATE.BG_3_HME_OPN_CMD;
      O     "CC_BUNKER_GATE_DB".BUNKER_GATE.BG_1_CLS_CMD;
      O     "CC_BUNKER_GATE_DB".BUNKER_GATE.BG_2_CLS_CMD;
      O     "CC_BUNKER_GATE_DB".BUNKER_GATE.BG_3_CLS_CMD;
      );
      A     "HALF_SECOND_PULSE_TRAIN";
      O     "MAIN_POWER_DB".LAMP_TEST_PB;
      );
      =     "CC_BUNKER_GATE_DB".BUNKER_GATE.BG_COAL_LD_PROG_IND;
END_FUNCTION

FUNCTION "OVEN_CHARGING_SF" : VOID	// FC 10
AUTHOR : Arun_Ram
VERSION : 0.1
BEGIN
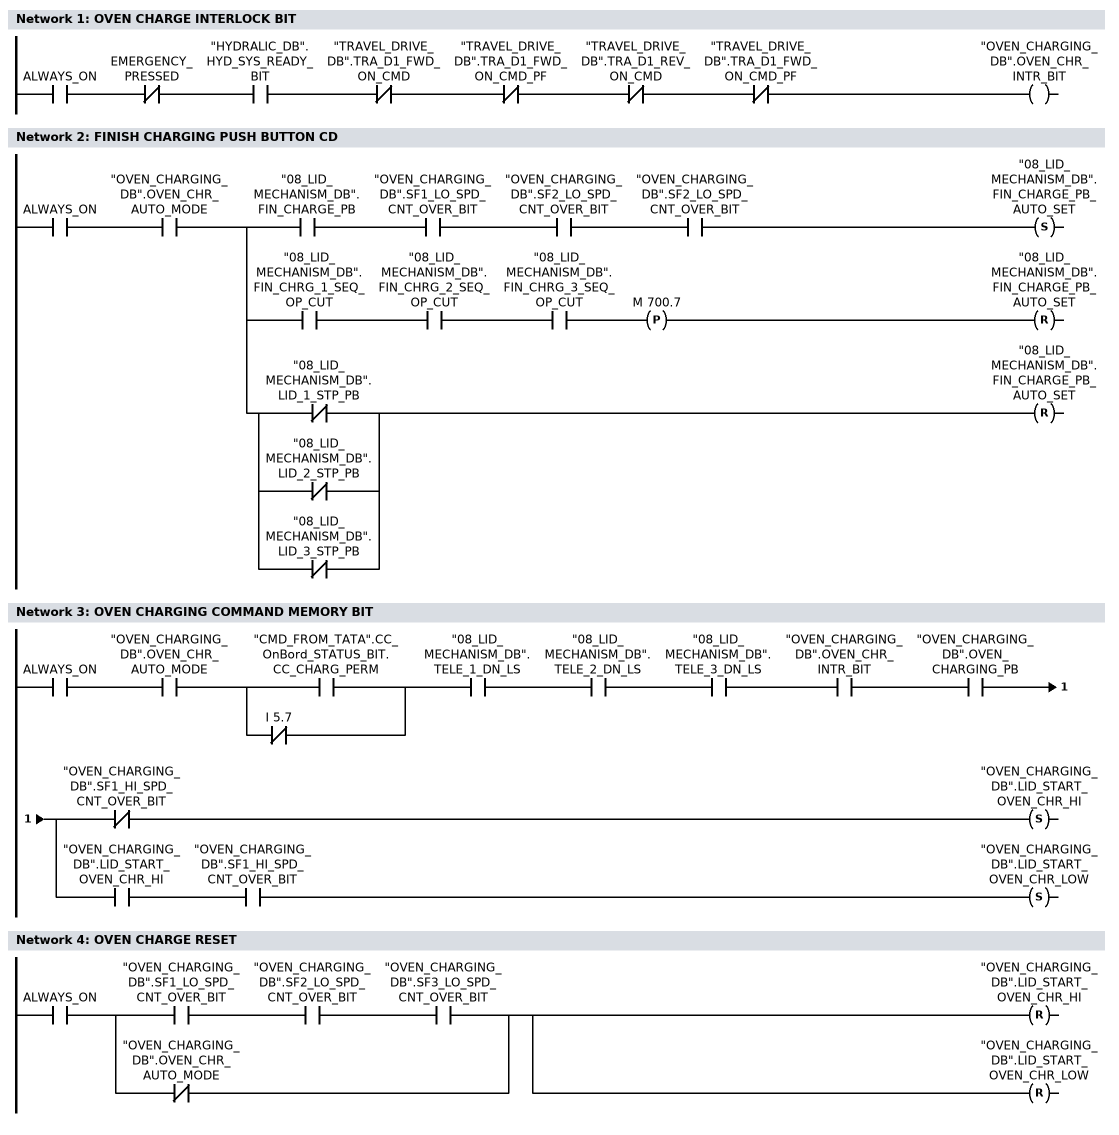
NETWORK
TITLE = OVEN CHARGE INTERLOCK BIT
      A     "ALWAYS_ON";
      AN    "EMERGENCY_PRESSED";
      A     "HYDRALIC_DB".HYD_SYS_READY_BIT;
      AN    "TRAVEL_DRIVE_DB".TRA_D1_FWD_ON_CMD;
      AN    "TRAVEL_DRIVE_DB".TRA_D1_FWD_ON_CMD_PF;
      AN    "TRAVEL_DRIVE_DB".TRA_D1_REV_ON_CMD;
      AN    "TRAVEL_DRIVE_DB".TRA_D1_FWD_ON_CMD_PF;
      =     "OVEN_CHARGING_DB".OVEN_CHR_INTR_BIT;
NETWORK
TITLE = FINISH CHARGING PUSH BUTTON CD
      A     "ALWAYS_ON";
      A     "OVEN_CHARGING_DB".OVEN_CHR_AUTO_MODE;
      =     L 0.0;
      A     L 0.0;
      A     "08_LID_MECHANISM_DB".FIN_CHARGE_PB;
      A     "OVEN_CHARGING_DB".SF1_LO_SPD_CNT_OVER_BIT;
      A     "OVEN_CHARGING_DB".SF2_LO_SPD_CNT_OVER_BIT;
      A     "OVEN_CHARGING_DB".SF2_LO_SPD_CNT_OVER_BIT;
      S     "08_LID_MECHANISM_DB".FIN_CHARGE_PB_AUTO_SET;
      A     L 0.0;
      A     "08_LID_MECHANISM_DB".FIN_CHRG_1_SEQ_OP_CUT;
      A     "08_LID_MECHANISM_DB".FIN_CHRG_2_SEQ_OP_CUT;
      A     "08_LID_MECHANISM_DB".FIN_CHRG_3_SEQ_OP_CUT;
      FP    M 700.7;
      R     "08_LID_MECHANISM_DB".FIN_CHARGE_PB_AUTO_SET;
      A     L 0.0;
      A(;
      ON    "08_LID_MECHANISM_DB".LID_1_STP_PB;
      ON    "08_LID_MECHANISM_DB".LID_2_STP_PB;
      ON    "08_LID_MECHANISM_DB".LID_3_STP_PB;
      );
      R     "08_LID_MECHANISM_DB".FIN_CHARGE_PB_AUTO_SET;
NETWORK
TITLE = OVEN CHARGING COMMAND MEMORY BIT
      A     "ALWAYS_ON";
      A     "OVEN_CHARGING_DB".OVEN_CHR_AUTO_MODE;
      A(;
      O     "CMD_FROM_TATA".CC_OnBord_STATUS_BIT.CC_CHARG_PERM;
      ON    I 5.7;
      );
      A     "08_LID_MECHANISM_DB".TELE_1_DN_LS;
      A     "08_LID_MECHANISM_DB".TELE_2_DN_LS;
      A     "08_LID_MECHANISM_DB".TELE_3_DN_LS;
      A     "OVEN_CHARGING_DB".OVEN_CHR_INTR_BIT;
      A     "OVEN_CHARGING_DB".OVEN_CHARGING_PB;
      =     L 0.0;
      A     L 0.0;
      AN    "OVEN_CHARGING_DB".SF1_HI_SPD_CNT_OVER_BIT;
      S     "OVEN_CHARGING_DB".LID_START_OVEN_CHR_HI;
      A     L 0.0;
      A     "OVEN_CHARGING_DB".LID_START_OVEN_CHR_HI;
      A     "OVEN_CHARGING_DB".SF1_HI_SPD_CNT_OVER_BIT;
      S     "OVEN_CHARGING_DB".LID_START_OVEN_CHR_LOW;
NETWORK
TITLE = OVEN CHARGE RESET
      A     "ALWAYS_ON";
      A(;
      A     "OVEN_CHARGING_DB".SF1_LO_SPD_CNT_OVER_BIT;
      A     "OVEN_CHARGING_DB".SF2_LO_SPD_CNT_OVER_BIT;
      A     "OVEN_CHARGING_DB".SF3_LO_SPD_CNT_OVER_BIT;
      ON    "OVEN_CHARGING_DB".OVEN_CHR_AUTO_MODE;
      );
      R     "OVEN_CHARGING_DB".LID_START_OVEN_CHR_HI;
      R     "OVEN_CHARGING_DB".LID_START_OVEN_CHR_LOW;
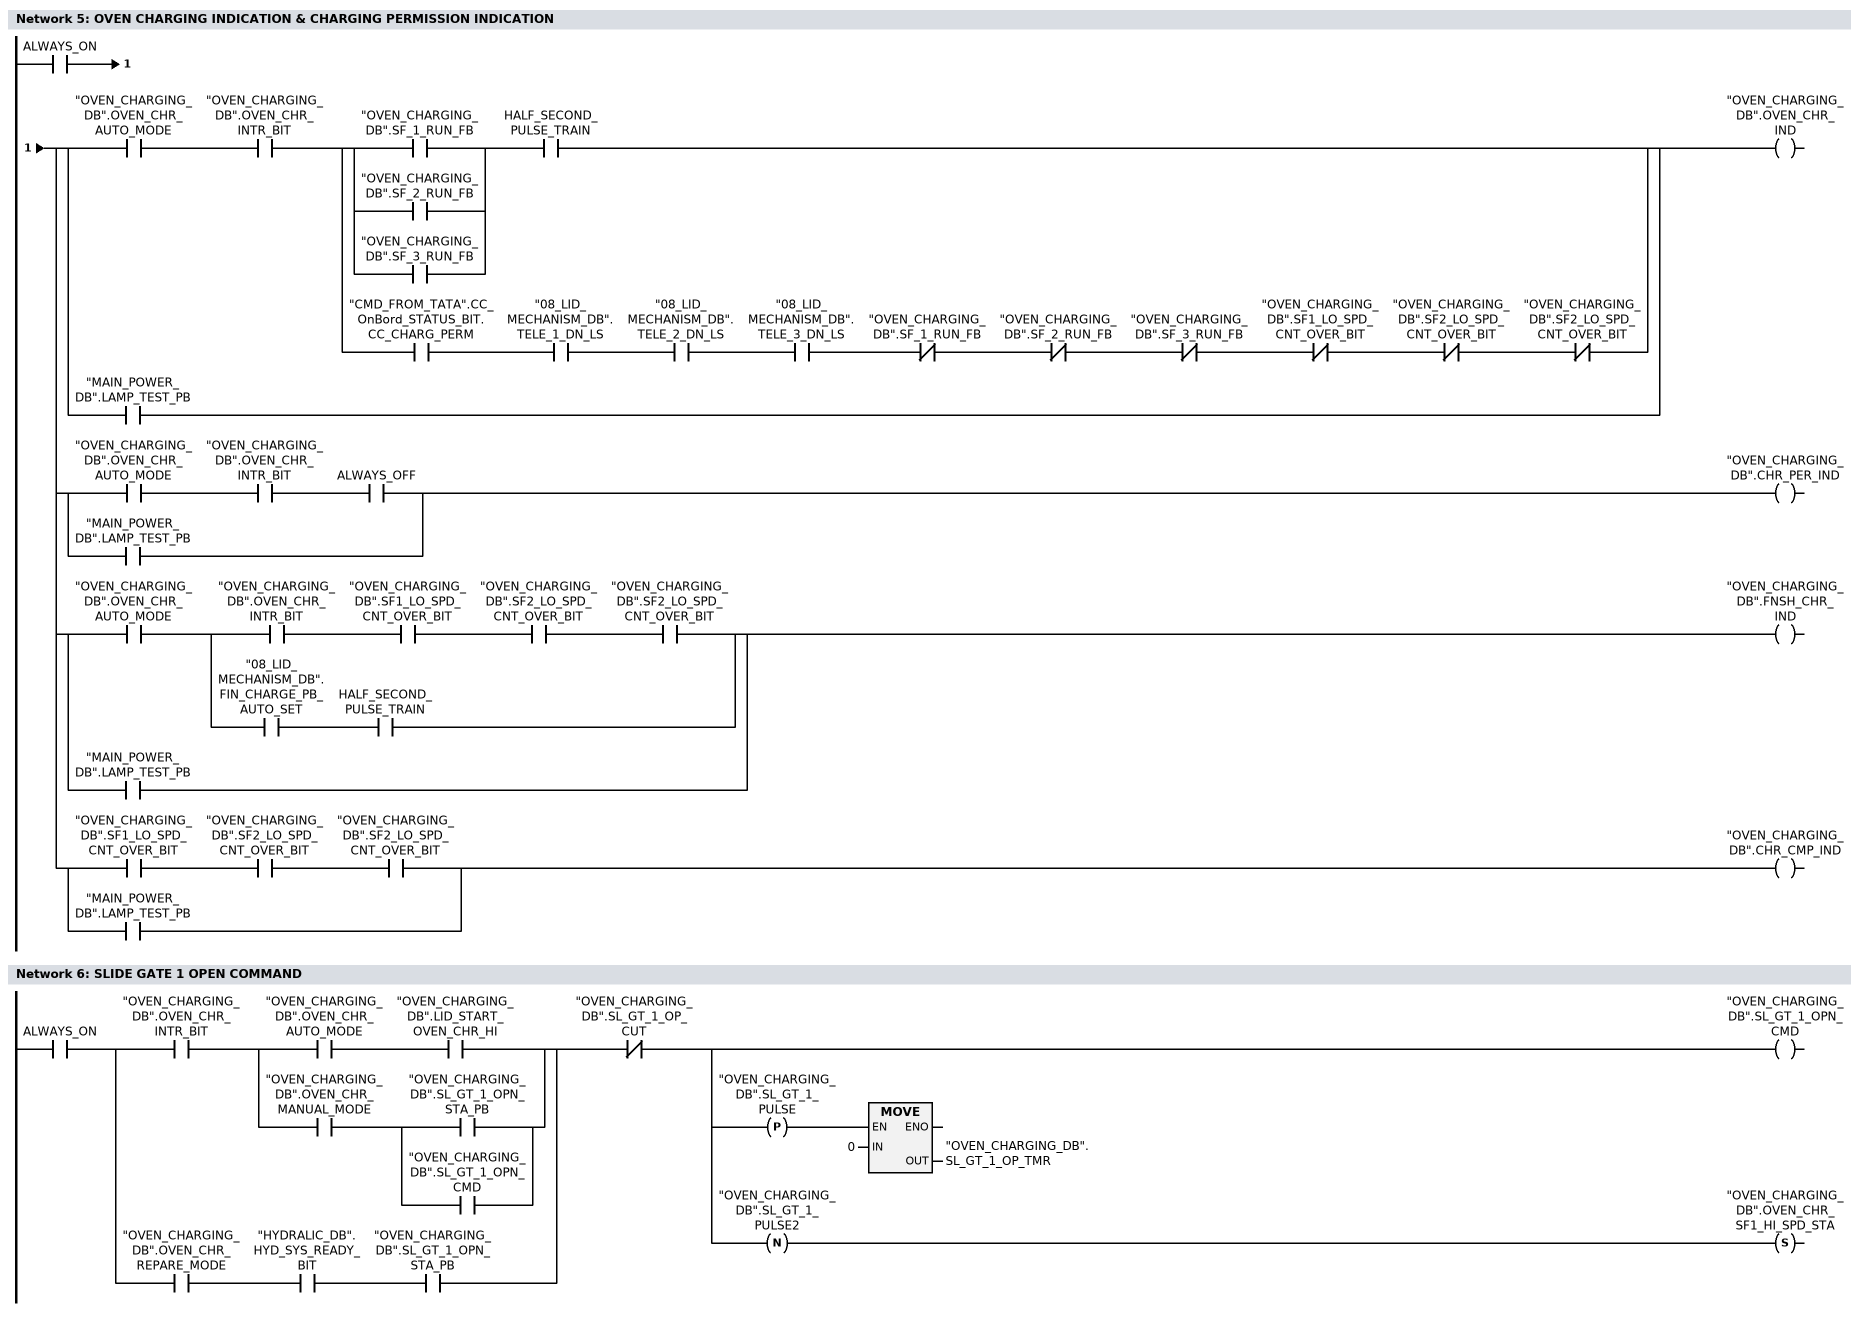
NETWORK
TITLE = OVEN CHARGING INDICATION & CHARGING PERMISSION INDICATION
      A     "ALWAYS_ON";
      =     L 0.0;
      A     L 0.0;
      A(;
      A     "OVEN_CHARGING_DB".OVEN_CHR_AUTO_MODE;
      A     "OVEN_CHARGING_DB".OVEN_CHR_INTR_BIT;
      A(;
      A(;
      O     "OVEN_CHARGING_DB".SF_1_RUN_FB;
      O     "OVEN_CHARGING_DB".SF_2_RUN_FB;
      O     "OVEN_CHARGING_DB".SF_3_RUN_FB;
      );
      A     "HALF_SECOND_PULSE_TRAIN";
      O;
      A     "CMD_FROM_TATA".CC_OnBord_STATUS_BIT.CC_CHARG_PERM;
      A     "08_LID_MECHANISM_DB".TELE_1_DN_LS;
      A     "08_LID_MECHANISM_DB".TELE_2_DN_LS;
      A     "08_LID_MECHANISM_DB".TELE_3_DN_LS;
      AN    "OVEN_CHARGING_DB".SF_1_RUN_FB;
      AN    "OVEN_CHARGING_DB".SF_2_RUN_FB;
      AN    "OVEN_CHARGING_DB".SF_3_RUN_FB;
      AN    "OVEN_CHARGING_DB".SF1_LO_SPD_CNT_OVER_BIT;
      AN    "OVEN_CHARGING_DB".SF2_LO_SPD_CNT_OVER_BIT;
      AN    "OVEN_CHARGING_DB".SF2_LO_SPD_CNT_OVER_BIT;
      );
      O     "MAIN_POWER_DB".LAMP_TEST_PB;
      );
      =     "OVEN_CHARGING_DB".OVEN_CHR_IND;
      A     L 0.0;
      A(;
      A     "OVEN_CHARGING_DB".OVEN_CHR_AUTO_MODE;
      A     "OVEN_CHARGING_DB".OVEN_CHR_INTR_BIT;
      A     "ALWAYS_OFF";
      O     "MAIN_POWER_DB".LAMP_TEST_PB;
      );
      =     "OVEN_CHARGING_DB".CHR_PER_IND;
      A     L 0.0;
      A(;
      A     "OVEN_CHARGING_DB".OVEN_CHR_AUTO_MODE;
      A(;
      A     "OVEN_CHARGING_DB".OVEN_CHR_INTR_BIT;
      A     "OVEN_CHARGING_DB".SF1_LO_SPD_CNT_OVER_BIT;
      A     "OVEN_CHARGING_DB".SF2_LO_SPD_CNT_OVER_BIT;
      A     "OVEN_CHARGING_DB".SF2_LO_SPD_CNT_OVER_BIT;
      O;
      A     "08_LID_MECHANISM_DB".FIN_CHARGE_PB_AUTO_SET;
      A     "HALF_SECOND_PULSE_TRAIN";
      );
      O     "MAIN_POWER_DB".LAMP_TEST_PB;
      );
      =     "OVEN_CHARGING_DB".FNSH_CHR_IND;
      A     L 0.0;
      A(;
      A     "OVEN_CHARGING_DB".SF1_LO_SPD_CNT_OVER_BIT;
      A     "OVEN_CHARGING_DB".SF2_LO_SPD_CNT_OVER_BIT;
      A     "OVEN_CHARGING_DB".SF2_LO_SPD_CNT_OVER_BIT;
      O     "MAIN_POWER_DB".LAMP_TEST_PB;
      );
      =     "OVEN_CHARGING_DB".CHR_CMP_IND;
NETWORK
TITLE = SLIDE GATE 1 OPEN COMMAND 
      A     "ALWAYS_ON";
      A(;
      A     "OVEN_CHARGING_DB".OVEN_CHR_INTR_BIT;
      A(;
      A     "OVEN_CHARGING_DB".OVEN_CHR_AUTO_MODE;
      A     "OVEN_CHARGING_DB".LID_START_OVEN_CHR_HI;
      O;
      A     "OVEN_CHARGING_DB".OVEN_CHR_MANUAL_MODE;
      A(;
      O     "OVEN_CHARGING_DB".SL_GT_1_OPN_STA_PB;
      O     "OVEN_CHARGING_DB".SL_GT_1_OPN_CMD;
      );
      );
      O;
      A     "OVEN_CHARGING_DB".OVEN_CHR_REPARE_MODE;
      A     "HYDRALIC_DB".HYD_SYS_READY_BIT;
      A     "OVEN_CHARGING_DB".SL_GT_1_OPN_STA_PB;
      );
      AN    "OVEN_CHARGING_DB".SL_GT_1_OP_CUT;
      =     L 0.0;
      A     L 0.0;
      BLD   102;
      =     "OVEN_CHARGING_DB".SL_GT_1_OPN_CMD;
      A     L 0.0;
      FP    "OVEN_CHARGING_DB".SL_GT_1_PULSE;
      JNB   _001;
      L     0;
      T     "OVEN_CHARGING_DB".SL_GT_1_OP_TMR;
_001: NOP   0;
      A     L 0.0;
      FN    "OVEN_CHARGING_DB".SL_GT_1_PULSE2;
      S     "OVEN_CHARGING_DB".OVEN_CHR_SF1_HI_SPD_STA;
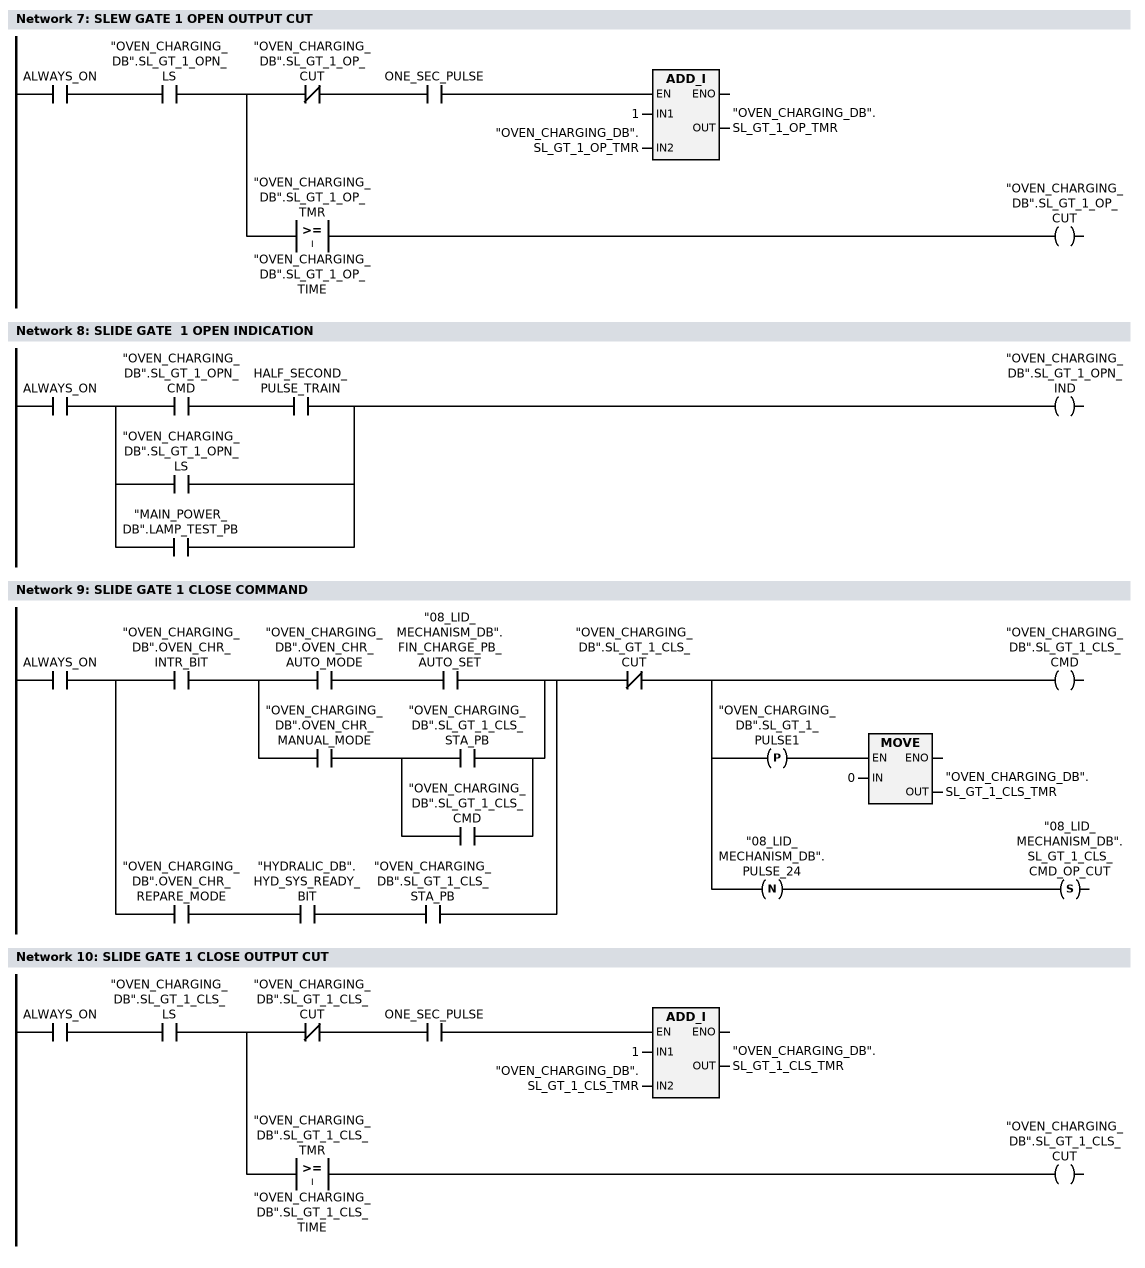
NETWORK
TITLE = SLEW GATE 1 OPEN OUTPUT CUT
      A     "ALWAYS_ON";
      A     "OVEN_CHARGING_DB".SL_GT_1_OPN_LS;
      =     L 0.0;
      A     L 0.0;
      AN    "OVEN_CHARGING_DB".SL_GT_1_OP_CUT;
      A     "ONE_SEC_PULSE";
      JNB   _002;
      L     1;
      L     "OVEN_CHARGING_DB".SL_GT_1_OP_TMR;
      +I;
      T     "OVEN_CHARGING_DB".SL_GT_1_OP_TMR;
_002: NOP   0;
      A     L 0.0;
      A(;
      L     "OVEN_CHARGING_DB".SL_GT_1_OP_TMR;
      L     "OVEN_CHARGING_DB".SL_GT_1_OP_TIME;
      >=I;
      );
      =     "OVEN_CHARGING_DB".SL_GT_1_OP_CUT;
NETWORK
TITLE = SLIDE GATE  1 OPEN INDICATION
      A     "ALWAYS_ON";
      A(;
      A     "OVEN_CHARGING_DB".SL_GT_1_OPN_CMD;
      A     "HALF_SECOND_PULSE_TRAIN";
      O     "OVEN_CHARGING_DB".SL_GT_1_OPN_LS;
      O     "MAIN_POWER_DB".LAMP_TEST_PB;
      );
      =     "OVEN_CHARGING_DB".SL_GT_1_OPN_IND;
NETWORK
TITLE = SLIDE GATE 1 CLOSE COMMAND
      A     "ALWAYS_ON";
      A(;
      A     "OVEN_CHARGING_DB".OVEN_CHR_INTR_BIT;
      A(;
      A     "OVEN_CHARGING_DB".OVEN_CHR_AUTO_MODE;
      A     "08_LID_MECHANISM_DB".FIN_CHARGE_PB_AUTO_SET;
      O;
      A     "OVEN_CHARGING_DB".OVEN_CHR_MANUAL_MODE;
      A(;
      O     "OVEN_CHARGING_DB".SL_GT_1_CLS_STA_PB;
      O     "OVEN_CHARGING_DB".SL_GT_1_CLS_CMD;
      );
      );
      O;
      A     "OVEN_CHARGING_DB".OVEN_CHR_REPARE_MODE;
      A     "HYDRALIC_DB".HYD_SYS_READY_BIT;
      A     "OVEN_CHARGING_DB".SL_GT_1_CLS_STA_PB;
      );
      AN    "OVEN_CHARGING_DB".SL_GT_1_CLS_CUT;
      =     L 0.0;
      A     L 0.0;
      BLD   102;
      =     "OVEN_CHARGING_DB".SL_GT_1_CLS_CMD;
      A     L 0.0;
      FP    "OVEN_CHARGING_DB".SL_GT_1_PULSE1;
      JNB   _003;
      L     0;
      T     "OVEN_CHARGING_DB".SL_GT_1_CLS_TMR;
_003: NOP   0;
      A     L 0.0;
      FN    "08_LID_MECHANISM_DB".PULSE_24;
      S     "08_LID_MECHANISM_DB".SL_GT_1_CLS_CMD_OP_CUT;
NETWORK
TITLE = SLIDE GATE 1 CLOSE OUTPUT CUT
      A     "ALWAYS_ON";
      A     "OVEN_CHARGING_DB".SL_GT_1_CLS_LS;
      =     L 0.0;
      A     L 0.0;
      AN    "OVEN_CHARGING_DB".SL_GT_1_CLS_CUT;
      A     "ONE_SEC_PULSE";
      JNB   _004;
      L     1;
      L     "OVEN_CHARGING_DB".SL_GT_1_CLS_TMR;
      +I;
      T     "OVEN_CHARGING_DB".SL_GT_1_CLS_TMR;
_004: NOP   0;
      A     L 0.0;
      A(;
      L     "OVEN_CHARGING_DB".SL_GT_1_CLS_TMR;
      L     "OVEN_CHARGING_DB".SL_GT_1_CLS_TIME;
      >=I;
      );
      =     "OVEN_CHARGING_DB".SL_GT_1_CLS_CUT;
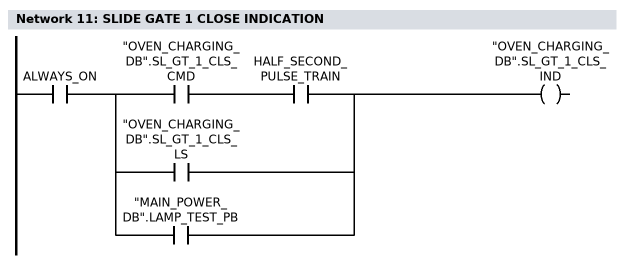
NETWORK
TITLE = SLIDE GATE 1 CLOSE INDICATION
      A     "ALWAYS_ON";
      A(;
      A     "OVEN_CHARGING_DB".SL_GT_1_CLS_CMD;
      A     "HALF_SECOND_PULSE_TRAIN";
      O     "OVEN_CHARGING_DB".SL_GT_1_CLS_LS;
      O     "MAIN_POWER_DB".LAMP_TEST_PB;
      );
      =     "OVEN_CHARGING_DB".SL_GT_1_CLS_IND;
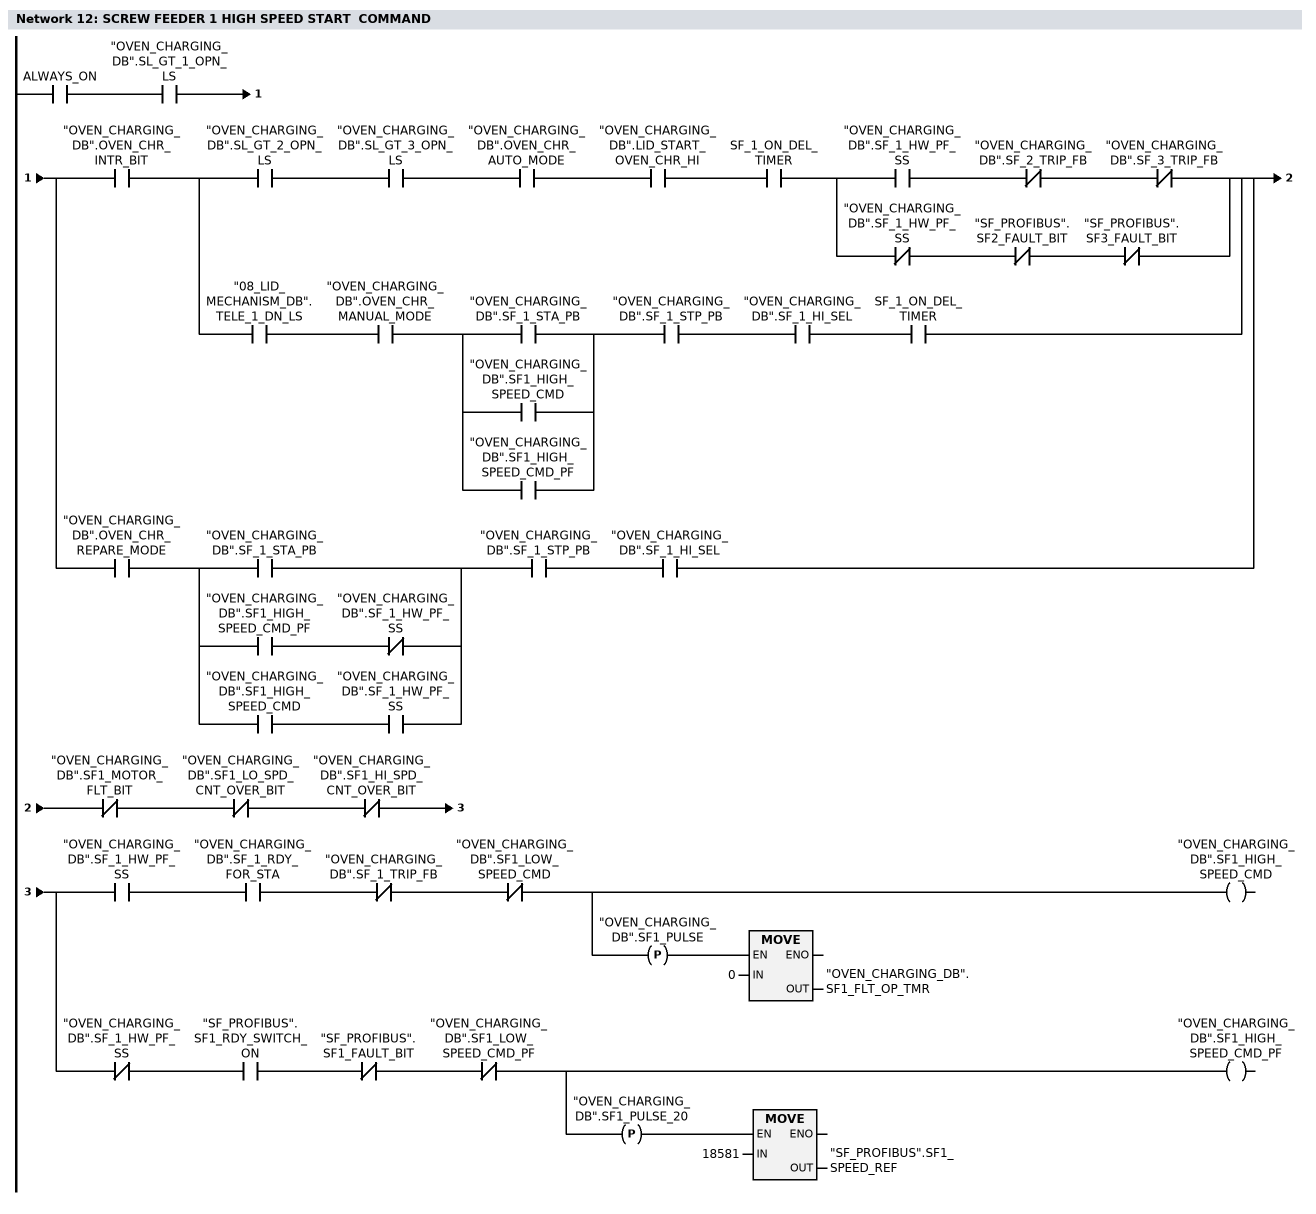
NETWORK
TITLE = SCREW FEEDER 1 HIGH SPEED START  COMMAND
      A     "ALWAYS_ON";
      A     "OVEN_CHARGING_DB".SL_GT_1_OPN_LS;
      A(;
      A     "OVEN_CHARGING_DB".OVEN_CHR_INTR_BIT;
      A(;
      A     "OVEN_CHARGING_DB".SL_GT_2_OPN_LS;
      A     "OVEN_CHARGING_DB".SL_GT_3_OPN_LS;
      A     "OVEN_CHARGING_DB".OVEN_CHR_AUTO_MODE;
      A     "OVEN_CHARGING_DB".LID_START_OVEN_CHR_HI;
      A     "SF_1_ON_DEL_TIMER";
      A(;
      A     "OVEN_CHARGING_DB".SF_1_HW_PF_SS;
      AN    "OVEN_CHARGING_DB".SF_2_TRIP_FB;
      AN    "OVEN_CHARGING_DB".SF_3_TRIP_FB;
      O;
      AN    "OVEN_CHARGING_DB".SF_1_HW_PF_SS;
      AN    "SF_PROFIBUS".SF2_FAULT_BIT;
      AN    "SF_PROFIBUS".SF3_FAULT_BIT;
      );
      O;
      A     "08_LID_MECHANISM_DB".TELE_1_DN_LS;
      A     "OVEN_CHARGING_DB".OVEN_CHR_MANUAL_MODE;
      A(;
      O     "OVEN_CHARGING_DB".SF_1_STA_PB;
      O     "OVEN_CHARGING_DB".SF1_HIGH_SPEED_CMD;
      O     "OVEN_CHARGING_DB".SF1_HIGH_SPEED_CMD_PF;
      );
      A     "OVEN_CHARGING_DB".SF_1_STP_PB;
      A     "OVEN_CHARGING_DB".SF_1_HI_SEL;
      A     "SF_1_ON_DEL_TIMER";
      );
      O;
      A     "OVEN_CHARGING_DB".OVEN_CHR_REPARE_MODE;
      A(;
      O     "OVEN_CHARGING_DB".SF_1_STA_PB;
      O;
      A     "OVEN_CHARGING_DB".SF1_HIGH_SPEED_CMD_PF;
      AN    "OVEN_CHARGING_DB".SF_1_HW_PF_SS;
      O;
      A     "OVEN_CHARGING_DB".SF1_HIGH_SPEED_CMD;
      A     "OVEN_CHARGING_DB".SF_1_HW_PF_SS;
      );
      A     "OVEN_CHARGING_DB".SF_1_STP_PB;
      A     "OVEN_CHARGING_DB".SF_1_HI_SEL;
      );
      AN    "OVEN_CHARGING_DB".SF1_MOTOR_FLT_BIT;
      AN    "OVEN_CHARGING_DB".SF1_LO_SPD_CNT_OVER_BIT;
      AN    "OVEN_CHARGING_DB".SF1_HI_SPD_CNT_OVER_BIT;
      =     L 0.0;
      A     L 0.0;
      A     "OVEN_CHARGING_DB".SF_1_HW_PF_SS;
      A     "OVEN_CHARGING_DB".SF_1_RDY_FOR_STA;
      AN    "OVEN_CHARGING_DB".SF_1_TRIP_FB;
      AN    "OVEN_CHARGING_DB".SF1_LOW_SPEED_CMD;
      =     L 0.1;
      A     L 0.1;
      BLD   102;
      =     "OVEN_CHARGING_DB".SF1_HIGH_SPEED_CMD;
      A     L 0.1;
      FP    "OVEN_CHARGING_DB".SF1_PULSE;
      JNB   _005;
      L     0;
      T     "OVEN_CHARGING_DB".SF1_FLT_OP_TMR;
_005: NOP   0;
      A     L 0.0;
      AN    "OVEN_CHARGING_DB".SF_1_HW_PF_SS;
      A     "SF_PROFIBUS".SF1_RDY_SWITCH_ON;
      AN    "SF_PROFIBUS".SF1_FAULT_BIT;
      AN    "OVEN_CHARGING_DB".SF1_LOW_SPEED_CMD_PF;
      =     L 0.1;
      A     L 0.1;
      BLD   102;
      =     "OVEN_CHARGING_DB".SF1_HIGH_SPEED_CMD_PF;
      A     L 0.1;
      FP    "OVEN_CHARGING_DB".SF1_PULSE_20;
      JNB   _006;
      L     18581;
      T     "SF_PROFIBUS".SF1_SPEED_REF;
_006: NOP   0;
